# B&R Automation Studio project NAELD004C00R10L518F00 (part 26)

#### Init.st
```iecst
(** 2019-05-20 **)
PROGRAM _INIT

	(* Always Change If Project Change *)

	//Pass Address To Global Address For External Use
	//Action, State & Status
	p_NtParamStat		:= ADR(eStat);
	p_NtParamStatus		:= ADR(eStatus);
	p_NtParamStatTxt	:= ADR(sStatTxt);

	//Alarm
	p_NtParamAlmData	:= ADR(tyAlmData);

	//Output
	p_NtParamFileNotFound				:= ADR(bFileNotFound);

	p_NtParamCurr						:= ADR(tyNtParamCurr);

	p_NtParamDISettings					:= ADR(tyNtParamCurr.tyDISettings);
	p_NtParamDOSettings					:= ADR(tyNtParamCurr.tyDOSettings);
	p_NtParamAWPusherPrep				:= ADR(tyNtParamCurr.bAWPusherPrep);
	p_NtParamAWPrep						:= ADR(tyNtParamCurr.bAWPrep);
	p_NtParamLFPrep						:= ADR(tyNtParamCurr.bLFPrep);
	p_NtParamLeaderMc					:= ADR(tyNtParamCurr.bLeaderMc);
	p_NtParamLFUsrSetPrep				:= ADR(tyNtParamCurr.bLFUsrSetPrep);
	p_NtParamLFWidthLimit				:= ADR(tyNtParamCurr.diLFWidthLimit);
	p_NtParamLFProdWidthChk				:= ADR(tyNtParamCurr.bLFProdWidthChk);
	p_NtParamDSWidthChkPrep				:= ADR(tyNtParamCurr.bDSWidthChkPrep);
	p_NtParamLCSLFPrep					:= ADR(tyNtParamCurr.bLCSLFPrep);
	p_NtParamLCSReqRcpPrep				:= ADR(tyNtParamCurr.bLCSReqRcpPrep);
	p_NtParamLCSManageRcpPrep			:= ADR(tyNtParamCurr.bLCSManageRcpPrep);
	p_NtParamLCSLiveDatPrep				:= ADR(tyNtParamCurr.bLCSLiveDatPrep);
	p_NtParamIPCSMEMA9851ExtdPrep		:= ADR(tyNtParamCurr.bIPCSMEMA9851ExtdPrep);
	p_NtParamVSMEMAPrep					:= ADR(tyNtParamCurr.bVSMEMAPrep);
	p_NtParamHermesPrep					:= ADR(tyNtParamCurr.bHermesPrep);
	p_NtParamHermesRmtPrep				:= ADR(tyNtParamCurr.bHermesRmtPrep);
	p_NtParamSSaverPrep					:= ADR(tyNtParamCurr.bSSaverPrep);
	p_NtParamWidthOffset				:= ADR(tyNtParamCurr.diWidthOffsetInUM);
	p_NtParamPushPulAWidthOffset		:= ADR(tyNtParamCurr.diAWPushPulOffsetInUM);
	p_NtParamJobNo						:= ADR(tyNtParamCurr.sJobNo);
	p_NtParamNtAddr						:= ADR(tyNtParamCurr.usiNtAddr);
	p_NtParamShutterWaitTmr				:= ADR(tyNtParamCurr.tShutterWaitTmr);
	p_NtParamProjAGVInPosSenPrep		:= ADR(tyNtParamCurr.bProjAGVInPosSenPrep);

	p_NtParamProjLaneBPrep				:= ADR(tyNtParamCurr.bProjLaneBPrep);
	p_NtParamProjTopToBtmDefault		:= ADR(tyNtParamCurr.bProjTopToBtmDefault);
	p_NtParamProjLongBrdPrep			:= ADR(tyNtParamCurr.bProjLongBrdPrep);
	p_NtParamProjInletShutPrep			:= ADR(tyNtParamCurr.bProjInletShutPrep);
	p_NtParamProjOutletShutPrep			:= ADR(tyNtParamCurr.bProjOutletShutPrep);
	p_NtParamProjMag1ConvPrep			:= ADR(tyNtParamCurr.bProjMag1ConvPrep);
	p_NtParamProjMag2ConvPrep			:= ADR(tyNtParamCurr.bProjMag2ConvPrep);
	p_NtParamProjMag3ConvPrep			:= ADR(tyNtParamCurr.bProjMag3ConvPrep);
	p_NtParamProjMag4ConvPrep			:= ADR(tyNtParamCurr.bProjMag4ConvPrep);
	p_NtParamProjMagOrientChkSenPrep	:= ADR(tyNtParamCurr.bProjMagOrientChkSenPrep);
	p_NtParamProjAGVPrep				:= ADR(tyNtParamCurr.bProjAGVPrep);
	p_NtParamProjBypsInitConvPrep		:= ADR(tyNtParamCurr.bProjBypsInitConvPrep);
	p_NtParamProjRlsNewProdPrep			:= ADR(tyNtParamCurr.bProjRlsNewProdPrep);
	p_NtParamProjBtnInsertRmvMag		:= ADR(tyNtParamCurr.bProjBtnInsertRmvMag);
	p_NtParamProjMagMinSlt				:= ADR(tyNtParamCurr.diProjMagMinSlt);
	p_NtParamProjMagMaxSlt				:= ADR(tyNtParamCurr.diProjMagMaxSlt);
	p_NtParamProjMag					:= ADR(tyNtParamCurr.eProjMag);
	p_NtParamProjConvDir				:= ADR(tyNtParamCurr.eProjConvDir);
	p_NtParamProjMagConvDir				:= ADR(tyNtParamCurr.eProjMagConvDir);
	p_NtParamProjMagAutoVerifyPrep		:= ADR(tyNtParamCurr.bMagAutoVerifyPrep);
	p_NtParamProjMotorizedPullerPrep	:= ADR(tyNtParamCurr.bProjMotorizedPullerPrep);
	p_NtParamProjMagSafetyBarPrep		:= ADR(tyNtParamCurr.bProjMagSafetyBarPrep);
	p_NtParamProjLifterMagPlatform		:= ADR(tyNtParamCurr.bProjLifterMagPlatform);

	p_NtParamUsrFolderProgNm			:= ADR(tyNtParamCurr.sUsrFolderProgNm);

	p_NtParamLibVersionProgNm			:= ADR(tyNtParamCurr.sLibVersionProgNm);

	p_NtParamTimeProgNm					:= ADR(tyNtParamCurr.sTimeProgNm);

	p_NtParamHWInfoProgNm				:= ADR(tyNtParamCurr.sHWInfoProgNm);
	p_NtParamHWInfoDevice				:= ADR(tyNtParamCurr.sHWInfoDevice);

	p_NtParamTLBuzMode					:= ADR(tyNtParamCurr.eTLBuzMode);

	p_NtParamTLChgRcpBlinkTm		:= ADR(tyNtParamCurr.tTLChgRcpBlinkTm);

	p_NtParamTLErrBlinkTm			:= ADR(tyNtParamCurr.tTLErrBlinkTm);
	p_NtParamBuzErrOnTm				:= ADR(tyNtParamCurr.tBuzErrOnTm);
	p_NtParamBuzErrRestTm			:= ADR(tyNtParamCurr.tBuzErrRestTm);
	p_NtParamBuzErrOnCntr			:= ADR(tyNtParamCurr.usiBuzErrOnCntr);
	p_NtParamBuzErrStopSeqEn		:= ADR(tyNtParamCurr.bBuzErrStopSeqEn);
	p_NtParamBuzErrStopSeqCntr		:= ADR(tyNtParamCurr.usiBuzErrStopSeqCntr);

	p_NtParamTLWarnBlinkTm			:= ADR(tyNtParamCurr.tTLWarnBlinkTm);
	p_NtParamBuzWarnOnTm			:= ADR(tyNtParamCurr.tBuzWarnOnTm);
	p_NtParamBuzWarnRestTm			:= ADR(tyNtParamCurr.tBuzWarnRestTm);
	p_NtParamBuzWarnOnCntr			:= ADR(tyNtParamCurr.usiBuzWarnOnCntr);
	p_NtParamBuzWarnStopSeqEn		:= ADR(tyNtParamCurr.bBuzWarnStopSeqEn);
	p_NtParamBuzWarnStopSeqCntr		:= ADR(tyNtParamCurr.usiBuzWarnStopSeqCntr);

	p_NtParamTLWarn1BlinkTm			:= ADR(tyNtParamCurr.tTLWarn1BlinkTm);
	p_NtParamBuzWarn1OnTm			:= ADR(tyNtParamCurr.tBuzWarn1OnTm);
	p_NtParamBuzWarn1RestTm			:= ADR(tyNtParamCurr.tBuzWarn1RestTm);
	p_NtParamBuzWarn1OnCntr			:= ADR(tyNtParamCurr.usiBuzWarn1OnCntr);
	p_NtParamBuzWarn1StopSeqEn		:= ADR(tyNtParamCurr.bBuzWarn1StopSeqEn);
	p_NtParamBuzWarn1StopSeqCntr	:= ADR(tyNtParamCurr.usiBuzWarn1StopSeqCntr);

	p_NtParamTLWarn2BlinkTm			:= ADR(tyNtParamCurr.tTLWarn2BlinkTm);
	p_NtParamBuzWarn2OnTm			:= ADR(tyNtParamCurr.tBuzWarn2OnTm);
	p_NtParamBuzWarn2RestTm			:= ADR(tyNtParamCurr.tBuzWarn2RestTm);
	p_NtParamBuzWarn2OnCntr			:= ADR(tyNtParamCurr.usiBuzWarn2OnCntr);
	p_NtParamBuzWarn2StopSeqEn		:= ADR(tyNtParamCurr.bBuzWarn2StopSeqEn);
	p_NtParamBuzWarn2StopSeqCntr	:= ADR(tyNtParamCurr.usiBuzWarn2StopSeqCntr);

	p_NtParamTLWarn3BlinkTm			:= ADR(tyNtParamCurr.tTLWarn3BlinkTm);
	p_NtParamBuzWarn3OnTm			:= ADR(tyNtParamCurr.tBuzWarn3OnTm);
	p_NtParamBuzWarn3RestTm			:= ADR(tyNtParamCurr.tBuzWarn3RestTm);
	p_NtParamBuzWarn3OnCntr			:= ADR(tyNtParamCurr.usiBuzWarn3OnCntr);
	p_NtParamBuzWarn3StopSeqEn		:= ADR(tyNtParamCurr.bBuzWarn3StopSeqEn);
	p_NtParamBuzWarn3StopSeqCntr	:= ADR(tyNtParamCurr.usiBuzWarn3StopSeqCntr);

	p_NtParamTLWarn4BlinkTm			:= ADR(tyNtParamCurr.tTLWarn4BlinkTm);
	p_NtParamBuzWarn4OnTm			:= ADR(tyNtParamCurr.tBuzWarn4OnTm);
	p_NtParamBuzWarn4RestTm			:= ADR(tyNtParamCurr.tBuzWarn4RestTm);
	p_NtParamBuzWarn4OnCntr			:= ADR(tyNtParamCurr.usiBuzWarn4OnCntr);
	p_NtParamBuzWarn4StopSeqEn		:= ADR(tyNtParamCurr.bBuzWarn4StopSeqEn);
	p_NtParamBuzWarn4StopSeqCntr	:= ADR(tyNtParamCurr.usiBuzWarn4StopSeqCntr);

	p_NtParamTLWarn5BlinkTm			:= ADR(tyNtParamCurr.tTLWarn5BlinkTm);
	p_NtParamBuzWarn5OnTm			:= ADR(tyNtParamCurr.tBuzWarn5OnTm);
	p_NtParamBuzWarn5RestTm			:= ADR(tyNtParamCurr.tBuzWarn5RestTm);
	p_NtParamBuzWarn5OnCntr			:= ADR(tyNtParamCurr.usiBuzWarn5OnCntr);
	p_NtParamBuzWarn5StopSeqEn		:= ADR(tyNtParamCurr.bBuzWarn5StopSeqEn);
	p_NtParamBuzWarn5StopSeqCntr	:= ADR(tyNtParamCurr.usiBuzWarn5StopSeqCntr);

	p_NtParamBuzAlertOnTm			:= ADR(tyNtParamCurr.tBuzAlertOnTm);
	p_NtParamBuzAlertRestTm			:= ADR(tyNtParamCurr.tBuzAlertRestTm);
	p_NtParamBuzAlertOnCntr			:= ADR(tyNtParamCurr.usiBuzAlertOnCntr);
	p_NtParamBuzAlertStopSeqEn		:= ADR(tyNtParamCurr.bBuzAlertStopSeqEn);
	p_NtParamBuzAlertStopSeqCntr	:= ADR(tyNtParamCurr.usiBuzAlertStopSeqCntr);

	p_NtParamTLBlueBlinkTm			:= ADR(tyNtParamCurr.tTLBlueBlinkTm);
	p_NtParamTLAmberBlinkTm			:= ADR(tyNtParamCurr.tTLAmberBlinkTm);
	p_NtParamTLWhiteBlinkTm			:= ADR(tyNtParamCurr.tTLWhiteBlinkTm);
	p_NtParamTLRedBlinkTm			:= ADR(tyNtParamCurr.tTLRedBlinkTm);
	p_NtParamTLGreenBlinkTm			:= ADR(tyNtParamCurr.tTLGreenBlinkTm);

	p_NtParamAlmProgNm					:= ADR(tyNtParamCurr.sAlmProgNm);
	p_NtParamAlmFileKeepDay				:= ADR(tyNtParamCurr.udiAlmFileKeepDay);

	p_NtParamProdRcpProgNm				:= ADR(tyNtParamCurr.sProdRcpProgNm);
	p_NtParamProdRcpListFileNm			:= ADR(tyNtParamCurr.sProdRcpListFileNm);
	p_NtParamProdRcpSingleFileNm		:= ADR(tyNtParamCurr.sProdRcpSingleFileNm);

	p_NtParamMpProdRcpProgNm			:= ADR(tyNtParamCurr.sMpProdRcpProgNm);
	p_NtParamMpProdRcpFileNm			:= ADR(tyNtParamCurr.sMpProdRcpFileNm);
	p_NtParamMpProdRcpPVNm				:= ADR(tyNtParamCurr.sMpProdRcpPVNm);

	p_NtParamMagRcpProgNm				:= ADR(tyNtParamCurr.sMagRcpProgNm);
	p_NtParamMagRcpListFileNm			:= ADR(tyNtParamCurr.sMagRcpListFileNm);
	p_NtParamMagRcpSingleFileNm			:= ADR(tyNtParamCurr.sMagRcpSingleFileNm);

	p_NtParamMagRcpProgNm1				:= ADR(tyNtParamCurr.sMagRcpProgNm1);
	p_NtParamMagRcpListFileNm1			:= ADR(tyNtParamCurr.sMagRcpListFileNm1);
	p_NtParamMagRcpSingleFileNm1		:= ADR(tyNtParamCurr.sMagRcpSingleFileNm1);

	p_NtParamMcParamProgNm				:= ADR(tyNtParamCurr.sMcParamProgNm);
	p_NtParamMcParamFileNm				:= ADR(tyNtParamCurr.sMcParamFileNm);

	p_NtParamUsrMgmtProgNm				:= ADR(tyNtParamCurr.sUsrMgmtProgNm);

	p_NtParamBffr1ProgNm				:= ADR(tyNtParamCurr.sBffr1ProgNm);
	p_NtParamBffr1FileNm				:= ADR(tyNtParamCurr.sBffr1FileNm);
	p_NtParamBffr1FIFO					:= ADR(tyNtParamCurr.bBffr1FIFO);

	p_NtParamBffr2ProgNm				:= ADR(tyNtParamCurr.sBffr2ProgNm);
	p_NtParamBffr2FileNm				:= ADR(tyNtParamCurr.sBffr2FileNm);
	p_NtParamBffr2FIFO					:= ADR(tyNtParamCurr.bBffr2FIFO);

	p_NtParamBffr3ProgNm				:= ADR(tyNtParamCurr.sBffr3ProgNm);
	p_NtParamBffr3FileNm				:= ADR(tyNtParamCurr.sBffr3FileNm);
	p_NtParamBffr3FIFO					:= ADR(tyNtParamCurr.bBffr3FIFO);

	p_NtParamBffr4ProgNm				:= ADR(tyNtParamCurr.sBffr4ProgNm);
	p_NtParamBffr4FileNm				:= ADR(tyNtParamCurr.sBffr4FileNm);
	p_NtParamBffr4FIFO					:= ADR(tyNtParamCurr.bBffr4FIFO);

	p_NtParamUSSMEMA1ProgNm				:= ADR(tyNtParamCurr.sUSSMEMA1ProgNm);
	p_NtParamUSSMEMA1RstDlyTm			:= ADR(tyNtParamCurr.tUSSMEMA1RstDlyTm);
	p_NtParamUSSMEMA1SigInChkTm			:= ADR(tyNtParamCurr.tUSSMEMA1SigInChkTm);

	p_NtParamUSSMEMA2ProgNm				:= ADR(tyNtParamCurr.sUSSMEMA2ProgNm);
	p_NtParamUSSMEMA2RstDlyTm			:= ADR(tyNtParamCurr.tUSSMEMA2RstDlyTm);
	p_NtParamUSSMEMA2SigInChkTm			:= ADR(tyNtParamCurr.tUSSMEMA2SigInChkTm);

	p_NtParamUSSMEMA3ProgNm				:= ADR(tyNtParamCurr.sUSSMEMA3ProgNm);
	p_NtParamUSSMEMA3RstDlyTm			:= ADR(tyNtParamCurr.tUSSMEMA3RstDlyTm);
	p_NtParamUSSMEMA3SigInChkTm			:= ADR(tyNtParamCurr.tUSSMEMA3SigInChkTm);

	p_NtParamUSSMEMA4ProgNm				:= ADR(tyNtParamCurr.sUSSMEMA4ProgNm);
	p_NtParamUSSMEMA4RstDlyTm			:= ADR(tyNtParamCurr.tUSSMEMA4RstDlyTm);
	p_NtParamUSSMEMA4SigInChkTm			:= ADR(tyNtParamCurr.tUSSMEMA4SigInChkTm);

	p_NtParamDSSMEMA1ProgNm				:= ADR(tyNtParamCurr.sDSSMEMA1ProgNm);
	p_NtParamDSSMEMA1RstDlyTm			:= ADR(tyNtParamCurr.tDSSMEMA1RstDlyTm);
	p_NtParamDSSMEMA1SigInChkTm			:= ADR(tyNtParamCurr.tDSSMEMA1SigInChkTm);

	p_NtParamDSSMEMA2ProgNm				:= ADR(tyNtParamCurr.sDSSMEMA2ProgNm);
	p_NtParamDSSMEMA2RstDlyTm			:= ADR(tyNtParamCurr.tDSSMEMA2RstDlyTm);
	p_NtParamDSSMEMA2SigInChkTm			:= ADR(tyNtParamCurr.tDSSMEMA2SigInChkTm);

	p_NtParamDSSMEMA3ProgNm				:= ADR(tyNtParamCurr.sDSSMEMA3ProgNm);
	p_NtParamDSSMEMA3RstDlyTm			:= ADR(tyNtParamCurr.tDSSMEMA3RstDlyTm);
	p_NtParamDSSMEMA3SigInChkTm			:= ADR(tyNtParamCurr.tDSSMEMA3SigInChkTm);

	p_NtParamDSSMEMA4ProgNm				:= ADR(tyNtParamCurr.sDSSMEMA4ProgNm);
	p_NtParamDSSMEMA4RstDlyTm			:= ADR(tyNtParamCurr.tDSSMEMA4RstDlyTm);
	p_NtParamDSSMEMA4SigInChkTm			:= ADR(tyNtParamCurr.tDSSMEMA4SigInChkTm);

	p_NtParamDSSMEMAAProgNm				:= ADR(tyNtParamCurr.sDSSMEMAAProgNm);
	p_NtParamDSSMEMAARstDlyTm			:= ADR(tyNtParamCurr.tDSSMEMAARstDlyTm);
	p_NtParamDSSMEMAASigInChkTm			:= ADR(tyNtParamCurr.tDSSMEMAASigInChkTm);

	p_NtParamDSSMEMABProgNm				:= ADR(tyNtParamCurr.sDSSMEMABProgNm);
	p_NtParamDSSMEMABRstDlyTm			:= ADR(tyNtParamCurr.tDSSMEMABRstDlyTm);
	p_NtParamDSSMEMABSigInChkTm			:= ADR(tyNtParamCurr.tDSSMEMABSigInChkTm);

	p_NtParamInShutterProgNm			:= ADR(tyNtParamCurr.sInShutterProgNm);
	p_NtParamInShutterTwoCtrlIn			:= ADR(tyNtParamCurr.bInShutterTwoCtrlIn);
	p_NtParamInShutterExtTO				:= ADR(tyNtParamCurr.tInShutterExtTO);
	p_NtParamInShutterRetTO				:= ADR(tyNtParamCurr.tInShutterRetTO);

	p_NtParamOutShutterProgNm			:= ADR(tyNtParamCurr.sOutShutterProgNm);
	p_NtParamOutShutterTwoCtrlIn		:= ADR(tyNtParamCurr.bOutShutterTwoCtrlIn);
	p_NtParamOutShutterExtTO			:= ADR(tyNtParamCurr.tOutShutterExtTO);
	p_NtParamOutShutterRetTO			:= ADR(tyNtParamCurr.tOutShutterRetTO);

	p_NtParamPullConvProgNm				:= ADR(tyNtParamCurr.sPullConvProgNm);
	p_NtParamPullConvOnDirMod			:= ADR(tyNtParamCurr.bPullConvOnDirMod);
	p_NtParamPullConvMtrOffDlyTm		:= ADR(tyNtParamCurr.tPullConvMtrOffDlyTm);
	p_NtParamPullConvPullExtTO			:= ADR(tyNtParamCurr.tPullConvPullExtTO);
	p_NtParamPullConvPullRetTO			:= ADR(tyNtParamCurr.tPullConvPullRetTO);
	p_NtParamPullConvRotHomeTO			:= ADR(tyNtParamCurr.tPullConvRotHomeTO);
	p_NtParamPullConvRotRemoteTO		:= ADR(tyNtParamCurr.tPullConvRotRemoteTO);

	p_NtParamMagConv1ProgNm				:= ADR(tyNtParamCurr.sMagConv1ProgNm);
	p_NtParamMagConv1OnDirMod			:= ADR(tyNtParamCurr.bMagConv1OnDirMod);
	p_NtParamMagConv1MtrOffDlyTm		:= ADR(tyNtParamCurr.tMagConv1MtrOffDlyTm);
	p_NtParamMagConv1ClprClampTO		:= ADR(tyNtParamCurr.tMagConv1ClprClampTO);
	p_NtParamMagConv1ClprUnclampTO		:= ADR(tyNtParamCurr.tMagConv1ClprUnclampTO);

	p_NtParamMagConv2ProgNm				:= ADR(tyNtParamCurr.sMagConv2ProgNm);
	p_NtParamMagConv2OnDirMod			:= ADR(tyNtParamCurr.bMagConv2OnDirMod);
	p_NtParamMagConv2MtrOffDlyTm		:= ADR(tyNtParamCurr.tMagConv2MtrOffDlyTm);
	p_NtParamMagConv2ClprClampTO		:= ADR(tyNtParamCurr.tMagConv2ClprClampTO);
	p_NtParamMagConv2ClprUnclampTO		:= ADR(tyNtParamCurr.tMagConv2ClprUnclampTO);

	p_NtParamMagConv3ProgNm				:= ADR(tyNtParamCurr.sMagConv3ProgNm);
	p_NtParamMagConv3OnDirMod			:= ADR(tyNtParamCurr.bMagConv3OnDirMod);
	p_NtParamMagConv3MtrOffDlyTm		:= ADR(tyNtParamCurr.tMagConv3MtrOffDlyTm);
	p_NtParamMagConv3ClprClampTO		:= ADR(tyNtParamCurr.tMagConv3ClprClampTO);
	p_NtParamMagConv3ClprUnclampTO		:= ADR(tyNtParamCurr.tMagConv3ClprUnclampTO);

	p_NtParamMagConv4ProgNm				:= ADR(tyNtParamCurr.sMagConv4ProgNm);
	p_NtParamMagConv4OnDirMod			:= ADR(tyNtParamCurr.bMagConv4OnDirMod);
	p_NtParamMagConv4MtrOffDlyTm		:= ADR(tyNtParamCurr.tMagConv4MtrOffDlyTm);
	p_NtParamMagConv4ClprClampTO		:= ADR(tyNtParamCurr.tMagConv4ClprClampTO);
	p_NtParamMagConv4ClprUnclampTO		:= ADR(tyNtParamCurr.tMagConv4ClprUnclampTO);

	p_NtParamMtrPshrProgNm				:= ADR(tyNtParamCurr.sMtrPshrProgNm);
	p_NtParamMtrPshrDir					:= ADR(tyNtParamCurr.bMtrPshrDir);
	p_NtParamMtrPshrAlmRstTm			:= ADR(tyNtParamCurr.tMtrPshrAlmRstTm);
	p_NtParamMtrPshrAlmTrigTm			:= ADR(tyNtParamCurr.tMtrPshrAlmTrigTm);
	p_NtParamMtrPshrExtTO				:= ADR(tyNtParamCurr.tMtrPshrExtTO);
	p_NtParamMtrPshrRetTO				:= ADR(tyNtParamCurr.tMtrPshrRetTO);
	p_NtParamMtrPshrExtSlowSpd			:= ADR(tyNtParamCurr.diMtrPshrExtSlowSpd);
	p_NtParamMtrPshrRetSlowSpd			:= ADR(tyNtParamCurr.diMtrPshrRetSlowSpd);
	p_NtParamMtrPshrExtNomSpd			:= ADR(tyNtParamCurr.diMtrPshrExtNomSpd);
	p_NtParamMtrPshrExtTorq				:= ADR(tyNtParamCurr.diMtrPshrExtTorq);
	p_NtParamMtrPshrRetTorq				:= ADR(tyNtParamCurr.diMtrPshrRetTorq);
	p_NtParamMtrPshrStartTorq			:= ADR(tyNtParamCurr.diMtrPshrStartTorq);

	p_NtParamAWPushPulProgNm			:= ADR(tyNtParamCurr.sAWPushPullProgNm);
	p_NtParamAWPushPulDevice			:= ADR(tyNtParamCurr.sAWPushPullDevice);
	p_NtParamAWPushPulNode				:= ADR(tyNtParamCurr.usiAWPushPullNode);
	p_NtParamAWPushPulDir				:= ADR(tyNtParamCurr.bAWPushPullDir);
	p_NtParamAWPushPulDirBl				:= ADR(tyNtParamCurr.bAWPushPullDirBl);
	p_NtParamAWPushPulPitchInUM			:= ADR(tyNtParamCurr.diAWPushPullPitchInUM);
	p_NtParamAWPushPulMovBlDistInUM		:= ADR(tyNtParamCurr.diAWPushPullMovBlDistInUM);
	p_NtParamAWPushPulParamInHm			:= ADR(tyNtParamCurr.tyAWPushPullParamInHm);
	p_NtParamAWPushPulParamInConvert	:= ADR(tyNtParamCurr.tyAWPushPullParamInConvert);
	p_NtParamAWPushPulParam				:= ADR(tyNtParamCurr.tyAWPushPullParam);
	p_NtParamAWPushPulAcc				:= ADR(tyNtParamCurr.tyAWPushPullParam.diAccInMS);
	p_NtParamAWPushPulDec				:= ADR(tyNtParamCurr.tyAWPushPullParam.diDecInMS);
	p_NtParamAWPushPulAutoSpd			:= ADR(tyNtParamCurr.tyAWPushPullParam.diAutoSpdInUMPS);
	p_NtParamAWPushPulTuning			:= ADR(tyNtParamCurr.tyAWPushPullTuning);
	p_NtParamAWPushPulMotorType			:= ADR(tyNtParamCurr.eAWPushPullServoMotorType);

	p_NtParamAWProgNm					:= ADR(tyNtParamCurr.sAWProgNm);
	p_NtParamAWDevice					:= ADR(tyNtParamCurr.sAWDevice);
	p_NtParamAWNode						:= ADR(tyNtParamCurr.usiAWNode);
	p_NtParamAWDir						:= ADR(tyNtParamCurr.bAWDir);
	p_NtParamAWDirBl					:= ADR(tyNtParamCurr.bAWDirBl);
	p_NtParamAWPitchInUM				:= ADR(tyNtParamCurr.diAWPitchInUM);
	p_NtParamAWMovBlDistInUM			:= ADR(tyNtParamCurr.diAWMovBlDistInUM);
	p_NtParamAWParamInHm				:= ADR(tyNtParamCurr.tyAWParamInHm);
	p_NtParamAWParamInConvert			:= ADR(tyNtParamCurr.tyAWParamInConvert);
	p_NtParamAWParam					:= ADR(tyNtParamCurr.tyAWParam);
	p_NtParamAWAcc						:= ADR(tyNtParamCurr.tyAWParam.diAccInMS);
	p_NtParamAWDec						:= ADR(tyNtParamCurr.tyAWParam.diDecInMS);
	p_NtParamAWAutoSpd					:= ADR(tyNtParamCurr.tyAWParam.diAutoSpdInUMPS);
	p_NtParamAWTuning					:= ADR(tyNtParamCurr.tyAWTuning);
	p_NtParamAWMotorType				:= ADR(tyNtParamCurr.eAWServoMotorType);

	p_NtParamTravProgNm					:= ADR(tyNtParamCurr.sTravProgNm);
	p_NtParamTravDevice					:= ADR(tyNtParamCurr.sTravDevice);
	p_NtParamTravNode					:= ADR(tyNtParamCurr.usiTravNode);
	p_NtParamTravDir					:= ADR(tyNtParamCurr.bTravDir);
	p_NtParamTravParamInHm				:= ADR(tyNtParamCurr.tyTravParamInHm);
	p_NtParamTravParamInConvert			:= ADR(tyNtParamCurr.tyTravParamInConvert);
	p_NtParamTravParam					:= ADR(tyNtParamCurr.tyTravParam);
	p_NtParamTravAcc					:= ADR(tyNtParamCurr.tyTravParam.diAccInMS);
	p_NtParamTravDec					:= ADR(tyNtParamCurr.tyTravParam.diDecInMS);
	p_NtParamTravAutoSpd				:= ADR(tyNtParamCurr.tyTravParam.diAutoSpdInUMPS);
	p_NtParamTravTuning					:= ADR(tyNtParamCurr.tyTravTuning);
	p_NtParamTravLongBrdAutoSpd			:= ADR(tyNtParamCurr.diTravAutoSpdLongBrdInUMPS);
	p_NtParamTravMotorType				:= ADR(tyNtParamCurr.eTravServoMotorType);

	p_NtParamLifterProgNm				:= ADR(tyNtParamCurr.sLifterProgNm);
	p_NtParamLifterDevice				:= ADR(tyNtParamCurr.sLifterDevice);
	p_NtParamLifterNode					:= ADR(tyNtParamCurr.usiLifterNode);
	p_NtParamLifterDir					:= ADR(tyNtParamCurr.bLifterDir);
	p_NtParamLifterParamInHm			:= ADR(tyNtParamCurr.tyLifterParamInHm);
	p_NtParamLifterParamInConvert		:= ADR(tyNtParamCurr.tyLifterParamInConvert);
	p_NtParamLifterParam				:= ADR(tyNtParamCurr.tyLifterParam);
	p_NtParamLifterAcc					:= ADR(tyNtParamCurr.tyLifterParam.diAccInMS);
	p_NtParamLifterDec					:= ADR(tyNtParamCurr.tyLifterParam.diDecInMS);
	p_NtParamLifterAutoSpd				:= ADR(tyNtParamCurr.tyLifterParam.diAutoSpdInUMPS);
	p_NtParamLifterTuning				:= ADR(tyNtParamCurr.tyLifterTuning);
	p_NtParamLifterMotorType			:= ADR(tyNtParamCurr.eLifterServoMotorType);

	p_NtParamDIProgNm					:= ADR(tyNtParamCurr.sDIProgNm);

	p_NtParamAIVSvrProgNm				:= ADR(tyNtParamCurr.sAGVSvrProgNm);

	p_NtParamAGVMag1ProgNm				:= ADR(tyNtParamCurr.sAGVMag1ProgNm);
	p_NtParamAGVMag2ProgNm				:= ADR(tyNtParamCurr.sAGVMag2ProgNm);
	p_NtParamAGVMag3ProgNm				:= ADR(tyNtParamCurr.sAGVMag3ProgNm);
	p_NtParamAGVMag4ProgNm				:= ADR(tyNtParamCurr.sAGVMag4ProgNm);

	p_NtParamHermesProgNm				:= ADR(tyNtParamCurr.sHermesProgNm);
	p_NtParamHermesRetainFileNm			:= ADR(tyNtParamCurr.sHermesRetainFileNm);
	p_NtParamHermesConfigFileNm			:= ADR(tyNtParamCurr.sHermesConfigFileNm);

	p_NtParamDSHermesAProgNm			:= ADR(tyNtParamCurr.sDSHermesAProgNm);
	p_NtParamDSHermesAFileKeepDay		:= ADR(tyNtParamCurr.udiDSHermesAFileKeepDay);
	p_NtParamDSHermesAAliveTmInSec		:= ADR(tyNtParamCurr.udiDSHermesAAliveTmInSec);
	p_NtParamDSHermesAConnTO			:= ADR(tyNtParamCurr.tDSHermesAConnTO);

	p_NtParamDSHermesBProgNm			:= ADR(tyNtParamCurr.sDSHermesBProgNm);
	p_NtParamDSHermesBFileKeepDay		:= ADR(tyNtParamCurr.udiDSHermesBFileKeepDay);
	p_NtParamDSHermesBAliveTmInSec		:= ADR(tyNtParamCurr.udiDSHermesBAliveTmInSec);
	p_NtParamDSHermesBConnTO			:= ADR(tyNtParamCurr.tDSHermesBConnTO);

	p_NtParamRmtHermesProgNm			:= ADR(tyNtParamCurr.sRmtHermesProgNm);
	p_NtParamRmtHermesConfigFileNm		:= ADR(tyNtParamCurr.sRmtHermesConfigFileNm);
	p_NtParamRmtHermesFileKeepDay		:= ADR(tyNtParamCurr.udiRmtHermesFileKeepDay);
	p_NtParamRmtHermesAliveTmInSec		:= ADR(tyNtParamCurr.udiRmtHermesAliveTmInSec);
	p_NtParamRmtHermesSndBffrSize		:= ADR(tyNtParamCurr.udiRmtHermesSndBffrSize);
	p_NtParamRmtHermesRcvBffrSize		:= ADR(tyNtParamCurr.udiRmtHermesRcvBffrSize);

	p_NtParamLFLeaderProgNm				:= ADR(tyNtParamCurr.sLFLeaderProgNm);
	p_NtParamLFLeaderOnlineChkDlyTm		:= ADR(tyNtParamCurr.tLFLeaderOnlineChkDlyTm);
	p_NtParamLFLeaderSetTmOffDlyTm		:= ADR(tyNtParamCurr.tLFLeaderSetTmOffDlyTm);

	p_NtParamLFFollowerProgNm			:= ADR(tyNtParamCurr.sLFFollowerProgNm);

	p_NtParamFollower1ProgNm			:= ADR(tyNtParamCurr.sFollower1ProgNm);
	p_NtParamFollower2ProgNm			:= ADR(tyNtParamCurr.sFollower2ProgNm);

	p_NtParamLCSProgNm					:= ADR(tyNtParamCurr.sLCSProgNm);

	p_NtParamLCSMngRcpProgNm			:= ADR(tyNtParamCurr.sLCSMngRcpProgNm);

	p_NtParamLCSLFProgNm				:= ADR(tyNtParamCurr.sLCSLFProgNm);

	p_NtParamOpsTravLifLDProgNm			:= ADR(tyNtParamCurr.sOpsTravLifLDProgNm);

	p_NtParamOpsMagLD1ProgNm			:= ADR(tyNtParamCurr.sOpsMagLD1ProgNm);

	p_NtParamOpsMagLD2ProgNm			:= ADR(tyNtParamCurr.sOpsMagLD2ProgNm);

	p_NtParamOpsMagLD3ProgNm			:= ADR(tyNtParamCurr.sOpsMagLD3ProgNm);

	p_NtParamOpsMagLD4ProgNm			:= ADR(tyNtParamCurr.sOpsMagLD4ProgNm);

	p_NtParamOpsMagConvLD1ProgNm		:= ADR(tyNtParamCurr.sOpsMagConvLD1ProgNm);

	p_NtParamOpsMagConvLD2ProgNm		:= ADR(tyNtParamCurr.sOpsMagConvLD2ProgNm);

	p_NtParamOpsMagConvLD3ProgNm		:= ADR(tyNtParamCurr.sOpsMagConvLD3ProgNm);

	p_NtParamOpsMagConvLD4ProgNm		:= ADR(tyNtParamCurr.sOpsMagConvLD4ProgNm);

	p_NtParamOpsLifMagLDProgNm			:= ADR(tyNtParamCurr.sOpsLifMagLDProgNm);

	p_NtParamProdRcpMinWidth			:= ADR(tyNtParamCurr.tyProdRcpWidth.diMin);
	p_NtParamProdRcpMaxWidth			:= ADR(tyNtParamCurr.tyProdRcpWidth.diMax);
	p_NtParamProdRcpMinMinSlt			:= ADR(tyNtParamCurr.tyProdRcpMinSlt.diMin);
	p_NtParamProdRcpMaxMinSlt			:= ADR(tyNtParamCurr.tyProdRcpMinSlt.diMax);
	p_NtParamProdRcpMinMaxSlt			:= ADR(tyNtParamCurr.tyProdRcpMaxSlt.diMin);
	p_NtParamProdRcpMaxMaxSlt			:= ADR(tyNtParamCurr.tyProdRcpMaxSlt.diMax);
	p_NtParamProdRcpMinPitch			:= ADR(tyNtParamCurr.tyProdRcpPitch.diMin);
	p_NtParamProdRcpMaxPitch			:= ADR(tyNtParamCurr.tyProdRcpPitch.diMax);
	p_NtParamProdRcpMinMcModA			:= ADR(tyNtParamCurr.tyProdRcpMcModA.diMin);
	p_NtParamProdRcpMaxMcModA			:= ADR(tyNtParamCurr.tyProdRcpMcModA.diMax);
	p_NtParamProdRcpMinMcModAB			:= ADR(tyNtParamCurr.tyProdRcpMcModAB.diMin);
	p_NtParamProdRcpMaxMcModAB			:= ADR(tyNtParamCurr.tyProdRcpMcModAB.diMax);

	p_NtParamPullerProgNm				:= ADR(tyNtParamCurr.sPullerProgNm);
	p_NtParamPullerTwoCtrlIn			:= ADR(tyNtParamCurr.bPullerTwoCtrlIn);
	p_NtParamPullerExtTO				:= ADR(tyNtParamCurr.tPullerExtTO);
	p_NtParamPullerRetTO				:= ADR(tyNtParamCurr.tPullerRetTO);
	p_NtParamProjPullerRotCylPrep		:= ADR(tyNtParamCurr.bProjPullerRotCylPrep);
	p_NtParamProjPullerExtMaxSlt		:= ADR(tyNtParamCurr.diProjPullerExtMaxSlt);
	p_NtParamProjPullerExtMinSlt		:= ADR(tyNtParamCurr.diProjPullerExtMinSlt);

	p_NtParamSelClamp1ProgNm			:= ADR(tyNtParamCurr.sSelClamp1ProgNm);
	p_NtParamSelClamp1TwoCtrlIn			:= ADR(tyNtParamCurr.bSelClamp1TwoCtrlIn);
	p_NtParamSelClamp1ExtDlyTm			:= ADR(tyNtParamCurr.tSelClamp1ExtDlyTm);
	p_NtParamSelClamp1RetDlyTm			:= ADR(tyNtParamCurr.tSelClamp1RetDlyTm);

	p_NtParamSelClamp2ProgNm			:= ADR(tyNtParamCurr.sSelClamp2ProgNm);
	p_NtParamSelClamp2TwoCtrlIn			:= ADR(tyNtParamCurr.bSelClamp2TwoCtrlIn);
	p_NtParamSelClamp2ExtDlyTm			:= ADR(tyNtParamCurr.tSelClamp2ExtDlyTm);
	p_NtParamSelClamp2RetDlyTm			:= ADR(tyNtParamCurr.tSelClamp2RetDlyTm);

	p_NtParamSelClamp3ProgNm			:= ADR(tyNtParamCurr.sSelClamp3ProgNm);
	p_NtParamSelClamp3TwoCtrlIn			:= ADR(tyNtParamCurr.bSelClamp3TwoCtrlIn);
	p_NtParamSelClamp3ExtDlyTm			:= ADR(tyNtParamCurr.tSelClamp3ExtDlyTm);
	p_NtParamSelClamp3RetDlyTm			:= ADR(tyNtParamCurr.tSelClamp3RetDlyTm);

	p_NtParamSelClamp4ProgNm			:= ADR(tyNtParamCurr.sSelClamp4ProgNm);
	p_NtParamSelClamp4TwoCtrlIn			:= ADR(tyNtParamCurr.bSelClamp4TwoCtrlIn);
	p_NtParamSelClamp4ExtDlyTm			:= ADR(tyNtParamCurr.tSelClamp4ExtDlyTm);
	p_NtParamSelClamp4RetDlyTm			:= ADR(tyNtParamCurr.tSelClamp4RetDlyTm);

	p_NtParamProjDBAOnRgtSen			:= ADR (tyNtParamCurr.bProjDBAOnRgtSen);

	p_NtParamLFWidth2Prep				:= ADR(tyNtParamCurr.bLFProdWidth2Prep);
	p_NtParamLFFllowerOnlineChkDlyTm	:= ADR(tyNtParamCurr.tLFFollowerOnlineChkDlyTm);

	p_NtParamUSSOT1ProgNm				:= ADR(tyNtParamCurr.sUSSOT1ProgNm);
	p_NtParamUSSOT1RstDlyTm				:= ADR(tyNtParamCurr.tUSSOT1RstDlyTm);
	p_NtParamUSSOT1SigInChkTm			:= ADR(tyNtParamCurr.tUSSOT1SigInChkTm);

	p_NtParamUSSOT2ProgNm				:= ADR(tyNtParamCurr.sUSSOT2ProgNm);
	p_NtParamUSSOT2RstDlyTm				:= ADR(tyNtParamCurr.tUSSOT2RstDlyTm);
	p_NtParamUSSOT2SigInChkTm			:= ADR(tyNtParamCurr.tUSSOT2SigInChkTm);

	p_NtParamUSSOT3ProgNm				:= ADR(tyNtParamCurr.sUSSOT3ProgNm);
	p_NtParamUSSOT3RstDlyTm				:= ADR(tyNtParamCurr.tUSSOT3RstDlyTm);
	p_NtParamUSSOT3SigInChkTm			:= ADR(tyNtParamCurr.tUSSOT3SigInChkTm);

	p_NtParamUSSOT4ProgNm				:= ADR(tyNtParamCurr.sUSSOT4ProgNm);
	p_NtParamUSSOT4RstDlyTm				:= ADR(tyNtParamCurr.tUSSOT4RstDlyTm);
	p_NtParamUSSOT4SigInChkTm			:= ADR(tyNtParamCurr.tUSSOT4SigInChkTm);

	p_NtParamDSSOT1ProgNm				:= ADR(tyNtParamCurr.sDSSOT1ProgNm);
	p_NtParamDSSOT1RstDlyTm				:= ADR(tyNtParamCurr.tDSSOT1RstDlyTm);
	p_NtParamDSSOT1SigInChkTm			:= ADR(tyNtParamCurr.tDSSOT1SigInChkTm);

	p_NtParamDSSOT2ProgNm				:= ADR(tyNtParamCurr.sDSSOT2ProgNm);
	p_NtParamDSSOT2RstDlyTm				:= ADR(tyNtParamCurr.tDSSOT2RstDlyTm);
	p_NtParamDSSOT2SigInChkTm			:= ADR(tyNtParamCurr.tDSSOT2SigInChkTm);

	p_NtParamDSSOT3ProgNm				:= ADR(tyNtParamCurr.sDSSOT3ProgNm);
	p_NtParamDSSOT3RstDlyTm				:= ADR(tyNtParamCurr.tDSSOT3RstDlyTm);
	p_NtParamDSSOT3SigInChkTm			:= ADR(tyNtParamCurr.tDSSOT3SigInChkTm);

	p_NtParamDSSOT4ProgNm				:= ADR(tyNtParamCurr.sDSSOT4ProgNm);
	p_NtParamDSSOT4RstDlyTm				:= ADR(tyNtParamCurr.tDSSOT4RstDlyTm);
	p_NtParamDSSOT4SigInChkTm			:= ADR(tyNtParamCurr.tDSSOT4SigInChkTm);

	p_NtParamProjSOTSenPrep				:= ADR(tyNtParamCurr.bProjSOTSensorPrep);

	p_NtParamMcProgNm					:= ADR(tyNtParamCurr.sMachineProgNm);
	p_NtParamMc1ProgNm					:= ADR(tyNtParamCurr.sMachine1ProgNm);

	p_NtParamProjUSBPrep				:= ADR(tyNtParamCurr.bUSBScannerPrep);
	p_NtParamUSBProgNm					:= ADR(tyNtParamCurr.sUSBRdrProgNm);

	p_NtParamSOTReadyOnFirst			:= ADR(tyNtParamCurr.bSOTReadyOnFirst);

	p_NtParamShowMESName				:= ADR(tyNtParamCurr.bShowMESName);
	p_NtParamShowFMorMESActive			:= ADR(tyNtParamCurr.bShowFMorMESActive);

	p_NtParamRS232Prep					:= ADR(tyNtParamCurr.bRS232ScannerPrep);
	p_NtParamRS232ProgNm				:= ADR(tyNtParamCurr.sRS232ProgNm);

	p_NtParamProdRcpMinMtrPshrExtSpd	:= ADR(tyNtParamCurr.tyProdRcpMtrPshrExtSpd.diMin);
	p_NtParamProdRcpMaxMtrPshrExtSpd	:= ADR(tyNtParamCurr.tyProdRcpMtrPshrExtSpd.diMax);
	p_NtParamProdRcpMinMtrPshrExtToq	:= ADR(tyNtParamCurr.tyProdRcpMtrPshrExtTorq.diMin);
	p_NtParamProdRcpMaxMtrPshrExtToq	:= ADR(tyNtParamCurr.tyProdRcpMtrPshrExtTorq.diMax);

	p_NtParamMag1SafetyBarProgNm		:= ADR(tyNtParamCurr.sMag1SafetyBarProgNm);
	p_NtParamMag1SafetyBarTwoCtrlIn		:= ADR(tyNtParamCurr.bMag1SafetyBarTwoCtrlIn);
	p_NtParamMag1SafetyBarExtTO			:= ADR(tyNtParamCurr.tMag1SafetyBarExtTO);
	p_NtParamMag1SafetyBarRetTO			:= ADR(tyNtParamCurr.tMag1SafetyBarRetTO);

	p_NtParamMag2SafetyBarProgNm		:= ADR(tyNtParamCurr.sMag2SafetyBarProgNm);
	p_NtParamMag2SafetyBarTwoCtrlIn		:= ADR(tyNtParamCurr.bMag2SafetyBarTwoCtrlIn);
	p_NtParamMag2SafetyBarExtTO			:= ADR(tyNtParamCurr.tMag2SafetyBarExtTO);
	p_NtParamMag2SafetyBarRetTO			:= ADR(tyNtParamCurr.tMag2SafetyBarRetTO);

	p_NtParamMag3SafetyBarProgNm		:= ADR(tyNtParamCurr.sMag3SafetyBarProgNm);
	p_NtParamMag3SafetyBarTwoCtrlIn		:= ADR(tyNtParamCurr.bMag3SafetyBarTwoCtrlIn);
	p_NtParamMag3SafetyBarExtTO			:= ADR(tyNtParamCurr.tMag3SafetyBarExtTO);
	p_NtParamMag3SafetyBarRetTO			:= ADR(tyNtParamCurr.tMag3SafetyBarRetTO);

	p_NtParamMag4SafetyBarProgNm		:= ADR(tyNtParamCurr.sMag4SafetyBarProgNm);
	p_NtParamMag4SafetyBarTwoCtrlIn		:= ADR(tyNtParamCurr.bMag4SafetyBarTwoCtrlIn);
	p_NtParamMag4SafetyBarExtTO			:= ADR(tyNtParamCurr.tMag4SafetyBarExtTO);
	p_NtParamMag4SafetyBarRetTO			:= ADR(tyNtParamCurr.tMag4SafetyBarRetTO);

	p_NtParamPullerHeightInMM			:= ADR(tyNtParamCurr.diPullerHeightInMM);

	p_NtParamProjDsFixToFixRail		:= ADR(tyNtParamCurr.bProjDSFixToFixRail);
	p_NtParamProjWorkOrderOPCUA		:= ADR(tyNtParamCurr.bProjWorkOrderOPCUA);

	p_NtParamProjServoPullPusherPrep	:= ADR(tyNtParamCurr.bProjServoPullerPusherPrep);
	p_NtParamPPProgNm					:= ADR(tyNtParamCurr.sPPProgNm);
	p_NtParamPPDevice					:= ADR(tyNtParamCurr.sPPDevice);
	p_NtParamPPNode						:= ADR(tyNtParamCurr.usiPPNode);
	p_NtParamPPDir						:= ADR(tyNtParamCurr.bPPDir);
	p_NtParamPPDirBl					:= ADR(tyNtParamCurr.bPPDirBl);
	p_NtParamPPPitchInUM				:= ADR(tyNtParamCurr.diPPPitchInUM);
	p_NtParamPPMovBlDistInUM			:= ADR(tyNtParamCurr.diPPMovBlDistInUM);
	p_NtParamPPParamInHm				:= ADR(tyNtParamCurr.tyPPParamInHm);
	p_NtParamPPParamInConvert			:= ADR(tyNtParamCurr.tyPPParamInConvert);
	p_NtParamPPParam					:= ADR(tyNtParamCurr.tyPPParam);
	p_NtParamPPAcc						:= ADR(tyNtParamCurr.tyPPParam.diAccInMS);
	p_NtParamPPDec						:= ADR(tyNtParamCurr.tyPPParam.diDecInMS);
	p_NtParamPPAutoSpd					:= ADR(tyNtParamCurr.tyPPParam.diAutoSpdInUMPS);
	p_NtParamPPTuning					:= ADR(tyNtParamCurr.tyPPTuning);
	p_NtParamPPMotorType				:= ADR(tyNtParamCurr.ePPServoMotorType);

	p_NtParamProjCurtainSenPrep			:= ADR(tyNtParamCurr.bProjCurtainSenPrep);
	p_NtParamProjMagHeightChkPrep		:= ADR(tyNtParamCurr.bProjMagHeightChkPrep);
	p_NtParamTravGotoMagWidthChkPt1		:= ADR(tyNtParamCurr.diTravGoToMagWidthChkPt1);
	p_NtParamTravGotoMagWidthChkPt2		:= ADR(tyNtParamCurr.diTravGoToMagWidthChkPt2);
	p_NtParamTravGotoMagWidthChkPt3		:= ADR(tyNtParamCurr.diTravGoToMagWidthChkPt3);

	p_NtParamPPTorqParam				:= ADR(tyNtParamCurr.tyPPTorqParam);
	p_NtParamProjLifTravMnlLoad			:= ADR(tyNtParamCurr.bProjLifTravMnlLoad);
	p_NtParamCustomerReq				:= ADR(tyNtParamCurr.eCustomerReq);
	p_NtParamProjShutter2Prep			:= ADR(tyNtParamCurr.bProjShutter2Prep);
	p_NtParamProjShutter3Prep			:= ADR(tyNtParamCurr.bProjShutter3Prep);

	//new for Hermes 1.3
	p_NtParamHermesSvyPrep			:= ADR(tyNtParamCurr.bHermesSvyPrep);
	p_NtParamHermesSvyFirstMc		:= ADR(tyNtParamCurr.bHermesSvyFirstMcInTheLine);//First Machine in the line, set for Loader / Destacker
	p_NtParamHermesSvyMagTypeMc		:= ADR(tyNtParamCurr.bHermesSvyMagTypeMc);//Magazine type Machine
	p_NtParamSvyHermesProgNm		:= ADR(tyNtParamCurr.sSvyHermesProgNm);
	p_NtParamSvyHermesConfigFileNm	:= ADR(tyNtParamCurr.sSvyHermesConfigFileNm);
	p_NtParamSvyHermesFileKeepDay	:= ADR(tyNtParamCurr.udiSvyHermesFileKeepDay);
	p_NtParamSvyHermesAliveTmInSec	:= ADR(tyNtParamCurr.udiSvyHermesAliveTmInSec);
	p_NtParamSvyHermesConnTO		:= ADR(tyNtParamCurr.tSvyHermesConnTO);
	p_NtParamSvyHermesRetainFileNm	:= ADR(tyNtParamCurr.sSvyHermesRetainFileNm);
	p_NtParamDSHermesRetainFileNm	:= ADR(tyNtParamCurr.sDSHermesRetainFileNm); //50 Board Data retain file name
	p_NtParamDSHermesMcCycleTm	    := ADR(tyNtParamCurr.rMachineCycleTime); //Machine Board Transfer Cycle Time
	p_NtParamDSHermesAWCycleTm	    := ADR(tyNtParamCurr.rAutoWidthCycleTime); //Machine Autowidth Cycle Time
	p_NtParamHermesScannerPrep    	:= ADR(tyNtParamCurr.bHermesScannerPrep);
	p_NtParamHermesInput            := ADR(tyNtParamCurr.iInput);//Total Input = How many inlet
	p_NtParamHermesOutput           := ADR(tyNtParamCurr.iOutput);//Total Outlet  = How many outlet

	p_NtParamAutoRcpPrep			:= ADR(tyNtParamCurr.bProjAutoRcpPrep);
	p_NtParamAutoRcpParamLmt		:= ADR(tyNtParamCurr.tyAutoRcpParamLmt);
	p_NtParamAutoRcpPrecededBy		:= ADR(tyNtParamCurr.eAutoRcpPrecededBy);

	//Add
	p_NtParmProjChinesePrep				:= ADR(tyNtParamCurr.bchineseprep);
	p_NtParmProjGermanPrep				:= ADR(tyNtParamCurr.bgermanprep);

	p_NtParamProjOutShutter2Prep	:= ADR(tyNtParamCurr.bProjOutShutter2Prep);
	p_NtParamProjCntrPullLmt		:= ADR(tyNtParamCurr.siProjCntrPullLmt);   //pull brd limit
	p_NtParamTrolleyLckPrep			:= ADR(tyNtParamCurr.bProjTrolleyLckPrep);
	p_NtParamTrolleyLckProgNm		:= ADR(tyNtParamCurr.sTrolleyLckProgNm);
	p_NtParamTrolleyLckTwoCtrlIn	:= ADR(tyNtParamCurr.bTrolleyLckTwoCtrlIn);
	p_NtParamTrolleyLckExtTO		:= ADR(tyNtParamCurr.tTrolleyLckExtTO);
	p_NtParamTrolleyLckRetTO		:= ADR(tyNtParamCurr.tTrolleyLckRetTO);

	p_NtParamTrolleyLckProgNm2		:= ADR(tyNtParamCurr.sTrolleyLckProgNm2);
	p_NtParamTrolleyLckTwoCtrlIn2	:= ADR(tyNtParamCurr.bTrolleyLckTwoCtrlIn2);
	p_NtParamTrolleyLckExtTO2		:= ADR(tyNtParamCurr.tTrolleyLckExtTO2);
	p_NtParamTrolleyLckRetTO2		:= ADR(tyNtParamCurr.tTrolleyLckRetTO2);

	(* Always Change If Project Change *)

END_PROGRAM
```

### Program Logical/UsrMgmt/UsrMgmt

#### Act_Alarm.st
```iecst
(** 2019-03-25 **)
ACTION Act_Alarm:

	//Error
	IF EDGEPOS(eStatus = Error) THEN

		tyAlmData.sProgNm		:= p_sProgNm;
		tyAlmData.udiCode		:= udiStatus;
		tyAlmData.eSeverity		:= AlmSeverityError;
		tyAlmData.udiRunTime	:= tyAlmData.udiRunTime + 1;
		tyAlmData.bAlm			:= TRUE;
		tyAlmData.udiModuleNum  := udiModuleNum;
		g_sUsrMgmtProgNm		:= p_sProgNm;
		//Get Error Message
		IF tyAlmData.udiCode < 10000 OR tyAlmData.udiCode > 10099 THEN
			tyAlmData.sAlmMsg	:= 'Unknown';
			tyAlmData.sRcyMsg	:= 'Unknown';
		ELSE
			tyAlmData.sAlmMsg	:= a_tyAlmText[tyAlmData.udiCode].sAlmText;
			tyAlmData.sRcyMsg	:= a_tyAlmText[tyAlmData.udiCode].sRcyText;
		END_IF

		sStatTxt	:= tyAlmData.sAlmMsg;

	ELSIF bRstErr AND (tyAlmData.udiCode <> 0) THEN

		tyAlmData.udiCode	:= 0;
		tyAlmData.eSeverity	:= AlmSeverityNA;
		tyAlmData.sAlmMsg	:= '';
		tyAlmData.sRcyMsg	:= '';
		tyAlmData.bAlm			:= FALSE;
		sStatTxt	:= a_sStatText[eStat];

	END_IF

END_ACTION
```

### Program Logical/Buffer/Buffer1 (IEC) - 1.00.0 - NtBuffer v5.00.0 , NtFileIO v5.00.0

#### InputRef_Link.var
```iecst
(*2019-04-09*)
(**)
(*External*)
VAR
	p_bLinkStartupRun : REFERENCE TO BOOL;
	p_bLinkNtParamProjMagConvPrep : REFERENCE TO BOOL;
	p_eLinkOpsMagLDBufferAct : REFERENCE TO eBufferAction;
	p_eLinkOpsMagConvLDBufferAct : REFERENCE TO eBufferAction;
END_VAR
(**)
VAR
	p_diLinkSltToSltDist : REFERENCE TO DINT;
	p_bLinkMcParamProdSelTopToBtm : REFERENCE TO BOOL;
	p_bLinkPresentSen1 : REFERENCE TO BOOL;
	p_bLinkPresentSen2 : REFERENCE TO BOOL;
END_VAR
(**)
VAR
	p_eLinkMag : REFERENCE TO eLDMag;
	p_usiLinkMod : REFERENCE TO USINT;
END_VAR
(**)
VAR
	p_diLinkMinSlt : REFERENCE TO DINT;
	p_diLinkMaxSlt : REFERENCE TO DINT;
	p_diLinkPitch : REFERENCE TO DINT;
	p_diLinkBffrTtlSlt : REFERENCE TO DINT;
	p_diLinkLifterBtmPosInUM : REFERENCE TO DINT;
END_VAR
(**)
VAR
	p_diLinkSltToSltDist1 : REFERENCE TO DINT;
	p_diLinkMinSlt1 : REFERENCE TO DINT;
	p_diLinkMaxSlt1 : REFERENCE TO DINT;
	p_diLinkPitch1 : REFERENCE TO DINT;
	p_diLinkBffrTtlSlt1 : REFERENCE TO DINT;
	p_diLinkLifterBtmPosInUM1 : REFERENCE TO DINT;
	p_bLinkNtParamProjRotCylPrep : REFERENCE TO BOOL;
END_VAR
(**)
VAR
	p_bLinkProjLifterMagPlatform : REFERENCE TO BOOL;
	p_diNtParamProjMagMaxSlt : REFERENCE TO DINT;
	p_eLinkOpsLifMagLDBufferAct : REFERENCE TO eBufferAction;
	p_bNtParamAutoRcpPrep : REFERENCE TO BOOL;
	p_bMcParamHermesSvyEn : REFERENCE TO BOOL;
	p_bHermesSvyPrep : REFERENCE TO BOOL;
	p_eNtParamCustomerReq : REFERENCE TO eCustomer;
	p_bMcParamMesRFIDEn : REFERENCE TO BOOL;
END_VAR
```

#### Act_InitGlobal.st
```iecst
(** 2019-04-26 **)
ACTION Act_InitGlobal:

	(* Always Change If Project Change *)

	//Pass Data To Link
	p_bLinkStartupRun ACCESS p_StartupRun;
	p_bLinkNtParamProjMagConvPrep ACCESS p_NtParamProjMag1ConvPrep;
//	p_eLinkOpsMagLDBufferAct ACCESS p_OpsMagLD1BufferAct;
	p_eLinkOpsMagConvLDBufferAct ACCESS p_OpsMagConvLD1BufferAct;

	p_bLinkMcParamProdSelTopToBtm ACCESS p_NtParamProjTopToBtmDefault;//p_ProdRcpCurrRcp1TopToBtm;
	p_bLinkPresentSen1 ACCESS p_DIMagPresentSen1;
	p_bLinkPresentSen2 ACCESS p_DIMagConvEntSen1;

	p_eLinkMag ACCESS p_NtParamProjMag;
	p_usiLinkMod ACCESS p_ProdRcpCurrRcp1McMod;

	p_diLinkSltToSltDist ACCESS p_MagRcpCurrRcpSltToSlt;
	p_diLinkMinSlt ACCESS p_ProdRcpCurrRcp1MinSltValue;
	p_diLinkMaxSlt ACCESS p_ProdRcpCurrRcp1MaxSltValue;
	p_diLinkPitch ACCESS p_ProdRcpCurrRcp1Pitch;
	p_diLinkBffrTtlSlt ACCESS p_MagRcpCurrRcpTtlSlt;
	p_diLinkLifterBtmPosInUM ACCESS p_MagRcpCurrRcpMag1Slt1Pos;

	p_diLinkSltToSltDist1 ACCESS p_MagRcpCurrRcpSltToSlt1;
	p_diLinkMinSlt1 ACCESS p_ProdRcpCurrRcp1MinSltRear;
	p_diLinkMaxSlt1 ACCESS p_ProdRcpCurrRcp1MaxSltRear;
	p_diLinkPitch1 ACCESS p_ProdRcpCurrRcp1PitchRear;
	p_diLinkBffrTtlSlt1 ACCESS p_MagRcpCurrRcpTtlSlt1;
	p_diLinkLifterBtmPosInUM1 ACCESS p_MagRcpCurrRcpMag1Slt1Pos1;

	p_bLinkNtParamProjRotCylPrep ACCESS p_NtParamProjPullerRotCylPrep;

	p_bLinkProjLifterMagPlatform ACCESS p_NtParamProjLifterMagPlatform;
	p_diNtParamProjMagMaxSlt ACCESS p_NtParamProjMagMaxSlt; //initial
	p_eLinkOpsLifMagLDBufferAct ACCESS p_OpsLifMagLDBufferAct1;
	p_bNtParamAutoRcpPrep ACCESS p_NtParamAutoRcpPrep;
	p_bHermesSvyPrep ACCESS p_NtParamHermesSvyPrep; //queryWO
	p_bMcParamHermesSvyEn ACCESS p_McParamHermesSvyEn;
	p_eNtParamCustomerReq ACCESS p_NtParamCustomerReq;
	p_bMcParamMesRFIDEn ACCESS p_McParamMesRFIDEn;

	//Pass Data To Internal Use
	p_udiRstErr ACCESS p_RstErrReset;
	p_sFileName ACCESS p_NtParamBffr1FileNm;
	p_bManual ACCESS p_UIMnlMod;
	p_dtCurrDT ACCESS p_TimeCurrDT;
//	p_diMinSlt ACCESS p_ProdRcpCurrRcp1MinSltValue;
//	p_diMaxSlt ACCESS p_ProdRcpCurrRcp1MaxSltValue;
//	p_diPitch ACCESS p_ProdRcpCurrRcp1Pitch;
//	p_diBffrTtlSlt ACCESS p_MagRcpCurrRcpTtlSlt;
//	p_diLifterBtmPosInUM ACCESS p_MagRcpCurrRcpMag1Slt1Pos;
	p_diLifterCurrPosInUM ACCESS p_LifterBtmActualPos;
	p_bFIFO ACCESS p_NtParamBffr1FIFO;
//	p_bMagPresentSensor ACCESS p_DIMagPresentSen1;
	p_sCurrRcpNm ACCESS p_ProdRcpCurrRcp1Nm;
	p_sProgNm ACCESS p_NtParamBffr1ProgNm;
	p_bNtSettingsLoadDone ACCESS p_StartupNtSettingsLoadDone;

	(* Always Change If Project Change *)

END_ACTION
```

#### Act_Initial.st
```iecst
(** 2019-04-26 **)
ACTION Act_Initial:

	//Initial
	sStatTxt	:= a_sStatText[eStat];

	fbDirCreate1.sDevice	:= 'F';
	fbDirCreate1.sDirName	:= 'User';
	fbDirCreate1(bEn := FALSE);

	fbDirCreate2.sDevice	:= 'User';
	fbDirCreate2.sDirName	:= 'Retain';
	fbDirCreate2(bEn := FALSE);

	fbFileRead1.sDevice			:= 'Retain';
	fbFileRead1.sFile			:= p_sFileName;
	fbFileRead1.udiOffset		:= 0;
	fbFileRead1.p_Dest			:= ADR(p_tyBuffer);
	fbFileRead1.udiLen			:= SIZEOF(p_tyBuffer);
	fbFileRead1(bEn := FALSE);

	fbFileWrite1.sDevice		:= 'Retain';
	fbFileWrite1.sFile			:= p_sFileName;
	fbFileWrite1.udiOffset		:= 0;
	fbFileWrite1.p_Src			:= ADR(p_tyBuffer);
	fbFileWrite1.udiLen			:= SIZEOF(p_tyBuffer);
	fbFileWrite1.udiOption		:= 0;
	fbFileWrite1(bEn := FALSE);

	fbCoolFanOffDlyTm.PT	:= DINT_TO_TIME(p_diCoolFanOffDlyTm);
	fbCoolFanOffDlyTm(IN := FALSE);

	fbCoolFanOffChkTm(IN := FALSE);
	fbMagAbsentTm(IN := FALSE);
	fbMagPresentTm(IN := FALSE);

	IF p_bLinkMcParamProdSelTopToBtm THEN
		diNxtUnloadSlt := 0;
	ELSE
		diNxtUnloadSlt := p_diNtParamProjMagMaxSlt;
	END_IF

END_ACTION
```

#### Act_Link.st
```iecst
(** 2019-03-29 **)
ACTION Act_Link:

	IF p_eLinkMag = LDMagQuadruple THEN
		CASE p_usiLinkMod OF
			0,2:  //LDModLoadLnA, LDModLoadLnAB:
				IF p_bAscending THEN
					p_diSltToSltInUM := p_diLinkSltToSltDist * -1;
				ELSE
					p_diSltToSltInUM := p_diLinkSltToSltDist;
				END_IF
				p_diMinSlt := p_diLinkMinSlt;
				p_diMaxSlt := p_diLinkMaxSlt;
				p_diPitch := p_diLinkPitch;
				p_diBffrTtlSlt := p_diLinkBffrTtlSlt;
				p_diLifterBtmPosInUM := p_diLinkLifterBtmPosInUM;

			1: //LDModLoadLnB:
				IF p_bAscending THEN
					p_diSltToSltInUM := p_diLinkSltToSltDist1 * -1;
				ELSE
					p_diSltToSltInUM := p_diLinkSltToSltDist1;
				END_IF
				p_diSltToSltInUM := p_diLinkSltToSltDist1;
				p_diMinSlt := p_diLinkMinSlt1;
				p_diMaxSlt := p_diLinkMaxSlt1;
				p_diPitch := p_diLinkPitch1;
				p_diBffrTtlSlt := p_diLinkBffrTtlSlt1;
				p_diLifterBtmPosInUM := p_diLinkLifterBtmPosInUM1;

		END_CASE
	ELSE

		IF p_bAscending THEN
			p_diSltToSltInUM := p_diLinkSltToSltDist * -1;
		ELSE
			p_diSltToSltInUM := p_diLinkSltToSltDist;
		END_IF
		IF p_bNtParamAutoRcpPrep AND ((p_bHermesSvyPrep AND p_bMcParamHermesSvyEn) OR (p_eNtParamCustomerReq = We_Fabricate AND p_bMcParamMesRFIDEn)) THEN
			p_diMinSlt ACCESS p_diAutoRcpMag1MinSlt;
			p_diMaxSlt ACCESS p_diAutoRcpMag1MaxSlt;
			p_diPitch ACCESS p_diAutoRcpMag1Pitch;
		ELSE
			p_diMinSlt ACCESS ADR(diMinSlt);
			p_diMaxSlt ACCESS ADR(diMaxSlt);
			p_diPitch ACCESS ADR(diPitch);
			p_diMinSlt := p_diLinkMinSlt;
			p_diMaxSlt := p_diLinkMaxSlt;
			p_diPitch := p_diLinkPitch;
		END_IF
		p_diBffrTtlSlt := p_diLinkBffrTtlSlt;
		p_diLifterBtmPosInUM := p_diLinkLifterBtmPosInUM;
	END_IF

	p_bAscending	:= NOT p_bLinkMcParamProdSelTopToBtm;
//	IF p_bLinkNtParamProjRotCylPrep THEN
//		p_bAscending := TRUE;
//	ELSE
//		p_bAscending := FALSE;
//	END_IF

	IF p_bLinkNtParamProjMagConvPrep THEN
		fbMagPresentTm.PT	:= T#2s;
	ELSE
		fbMagPresentTm.PT	:= T#8s;
	END_IF

	p_bMagPresentSensor := p_bLinkPresentSen1 OR p_bLinkPresentSen2;

END_ACTION
```

#### Act_LinkAction.st
```iecst
(** 2019-05-10 **)
ACTION Act_LinkAction:

	IF p_bLinkStartupRun = TRUE THEN
		p_eAct ACCESS p_StartupBuffer1Act;
	ELSE
		IF eStatus = Idle THEN
			IF p_bLinkProjLifterMagPlatform = FALSE THEN
				IF p_eLinkOpsMagConvLDBufferAct <> BufferActIdle THEN
					p_eAct ACCESS p_OpsMagConvLD1BufferAct;
				ELSE
					p_eAct ACCESS p_UIBuffer1Act;
				END_IF
			ELSE
				IF p_eLinkOpsLifMagLDBufferAct <> BufferActIdle THEN
					p_eAct ACCESS p_OpsLifMagLDBufferAct1;
				ELSE
					p_eAct ACCESS p_UIBuffer1Act;
				END_IF
			END_IF
		END_IF
	END_IF

END_ACTION
```

#### Act_Main.st
```iecst
(** 2019-07-03 **)
ACTION Act_Main:

	IF eStatOld <> eStat THEN
		fbDirCreate1(bEn := FALSE);
		fbDirCreate2(bEn := FALSE);
		fbFileRead1(bEn := FALSE);
		fbFileWrite1(bEn := FALSE);
		usiStep	:= 0;

		bFileNotFound			:= FALSE;
		bNewProduct				:= FALSE;
		bLastProductUnload		:= FALSE;
		bLastProductLeftInBffr	:= FALSE;

		sStatTxt	:= a_sStatText[eStat];

		eStatOld	:= eStat;

		eStatus		:= Busy;
	END_IF

	//Main
	CASE eStat OF

		BufferActIdle:
			eStatus	:= Idle;

		BufferActCreateDir:
			IF eStatus = Idle OR eStatus = Busy THEN

				eStatus	:= Busy;

				CASE usiStep OF
					0:
						fbDirCreate1(bEn := TRUE);
						IF fbDirCreate1.udiStatus = 0 THEN
							usiStep	:= 1;
						ELSIF fbDirCreate1.udiStatus < 65534 THEN
							eStatus		:= Error;

							IF fbDirCreate1.udiStatus = 1908 THEN
								udiStatus	:= 10000;	//Create User Directory Error
							ELSE
								udiStatus	:= fbDirCreate1.udiStatus;
							END_IF
						END_IF

					1:
						fbDirCreate2(bEn := TRUE);
						IF fbDirCreate2.udiStatus = 0 THEN
							eStatus	:= Done;
						ELSIF fbDirCreate2.udiStatus < 65534 THEN
							eStatus		:= Error;

							IF fbDirCreate2.udiStatus = 1908 THEN
								udiStatus	:= 10001;	//Create Retain Directory Error
							ELSE
								udiStatus	:= fbDirCreate2.udiStatus;
							END_IF
						END_IF

				END_CASE

			END_IF

		BufferActGetRetainBffr:
			IF eStatus = Idle OR eStatus = Busy THEN

				eStatus	:= Busy;

				fbFileRead1(bEn := TRUE);
				IF fbFileRead1.udiStatus = 0 THEN
					eStatus	:= Done;

					tyBffrParameter.diBffrTtlSlt	:= p_diBffrTtlSlt;
					tyBffrParameter.diSltCap		:= p_diSltCap;

					fBffrStat(ADR(p_tyBufferStat) , p_tyBuffer);
					fDispBffrDescending(ADR(p_tyDispBuffer) , tyBffrParameter , p_tyBuffer , p_dtCurrDT , DINT_TO_TIME(p_diCoolTm) , 0 , 1 , 2);

				ELSIF fbFileRead1.udiStatus < 65534 THEN
					eStatus	:= Error;

					IF fbFileRead1.udiStatus = 1900 THEN
						udiStatus	:= 10002;	//File Open Error While Reading Retain File
					ELSIF fbFileRead1.udiStatus = 1902 THEN
						udiStatus	:= 10003;	//File Read Error While Reading Retain File
					ELSIF fbFileRead1.udiStatus = 1904 THEN
						udiStatus	:= 10004;	//File Close Error While Reading Retain File
					ELSIF fbFileRead1.udiStatus = 1915 THEN
						eStatus			:= Done;
						bFileNotFound	:= TRUE;
					ELSE
						udiStatus	:= fbFileRead1.udiStatus;
					END_IF
				END_IF

			END_IF

		BufferActSetFull:
			IF eStatus = Idle OR eStatus = Busy THEN

				eStatus	:= Busy;

				CASE usiStep OF
					0:
						tyBffrParameter.bAscending		:= p_bAscending;
						tyBffrParameter.diBffrTtlSlt	:= p_diBffrTtlSlt;
						tyBffrParameter.diMaxSlt		:= p_diMaxSlt;
						tyBffrParameter.diMinSlt		:= p_diMinSlt;
						tyBffrParameter.diPitch			:= p_diPitch;
						tyBffrParameter.diSltCap		:= p_diSltCap;
						tyBffrParameter.a_bSkip			:= pa_bSkip;
						bFIFOOld						:= p_bFIFO;

						udiStatus	:= fBffrSetFull(ADR(p_tyBuffer) , tyBffrParameter , p_dtCurrDT , p_sBffrNm , p_sProdNm);

						IF udiStatus = 0 THEN
							usiStep	:= 1;

							fBffrStat(ADR(p_tyBufferStat) , p_tyBuffer);
							fDispBffrDescending(ADR(p_tyDispBuffer) , tyBffrParameter , p_tyBuffer , p_dtCurrDT , DINT_TO_TIME(p_diCoolTm) , 0 , 1 , 2);

						ELSE
							eStatus	:= Error;

						END_IF

					1:
						fbFileWrite1(bEn := TRUE);

						IF fbFileWrite1.udiStatus = 0 THEN
							eStatus	:= Done;
						ELSIF fbFileWrite1.udiStatus < 65534 THEN
							eStatus	:= Error;

							IF fbFileWrite1.udiStatus = 1900 THEN
								udiStatus	:= 10005;	//File Open Error While Setting Full Buffer
							ELSIF fbFileWrite1.udiStatus = 1901 THEN
								udiStatus	:= 10006;	//File Create Error While Setting Full Buffer
							ELSIF fbFileWrite1.udiStatus = 1903 THEN
								udiStatus	:= 10007;	//File Write Error While Setting Full Buffer
							ELSIF fbFileWrite1.udiStatus = 1904 THEN
								udiStatus	:= 10008;	//File Close Error While Setting Full Buffer
							ELSIF fbFileWrite1.udiStatus = 1914 THEN
								udiStatus	:= 10040;	//Directory Does Not Exist While Setting Full Buffer
							ELSE
								udiStatus	:= fbFileWrite1.udiStatus;
							END_IF
						END_IF

				END_CASE

			END_IF

		BufferActSetMty:
			IF eStatus = Idle OR eStatus = Busy THEN

				eStatus	:= Busy;

				CASE usiStep OF
					0:
						tyBffrParameter.bAscending		:= p_bAscending;
						tyBffrParameter.diBffrTtlSlt	:= p_diBffrTtlSlt;
						tyBffrParameter.diMaxSlt		:= p_diMaxSlt;
						tyBffrParameter.diMinSlt		:= p_diMinSlt;
						tyBffrParameter.diPitch			:= p_diPitch;
						tyBffrParameter.diSltCap		:= p_diSltCap;
						tyBffrParameter.a_bSkip			:= pa_bSkip;
						bFIFOOld						:= p_bFIFO;

						udiStatus	:= fBffrSetMty(ADR(p_tyBuffer) , tyBffrParameter , p_sBffrNm);

						IF udiStatus = 0 THEN
							usiStep	:= 1;

							fBffrStat(ADR(p_tyBufferStat) , p_tyBuffer);
							fDispBffrDescending(ADR(p_tyDispBuffer) , tyBffrParameter , p_tyBuffer , p_dtCurrDT , DINT_TO_TIME(p_diCoolTm) , 0 , 1 , 2);

						ELSE
							eStatus	:= Error;

						END_IF

					1:
						fbFileWrite1(bEn := TRUE);

						IF fbFileWrite1.udiStatus = 0 THEN
							eStatus	:= Done;
						ELSIF fbFileWrite1.udiStatus < 65534 THEN
							eStatus	:= Error;

							IF fbFileWrite1.udiStatus = 1900 THEN
								udiStatus	:= 10009;	//File Open Error While Setting Empty Buffer
							ELSIF fbFileWrite1.udiStatus = 1901 THEN
								udiStatus	:= 10010;	//File Create Error While Setting Empty Buffer
							ELSIF fbFileWrite1.udiStatus = 1903 THEN
								udiStatus	:= 10011;	//File Write Error While Setting Empty Buffer
							ELSIF fbFileWrite1.udiStatus = 1904 THEN
								udiStatus	:= 10012;	//File Close Error While Setting Empty Buffer
							ELSIF fbFileWrite1.udiStatus = 1914 THEN
								udiStatus	:= 10041;	//Directory Does Not Exist While Setting Empty Buffer
							ELSE
								udiStatus	:= fbFileWrite1.udiStatus;
							END_IF
						END_IF

				END_CASE

			END_IF

		BufferActLoad:
			IF eStatus = Idle OR eStatus = Busy THEN

				eStatus	:= Busy;

				CASE usiStep OF
					0:
						diCurrSlt	:= fLifterPosInUMToSltBtmMin(p_diLifterCurrPosInUM , p_diSltToSltInUM , p_diLifterBtmPosInUM);

						udiStatus	:= fBffrLoad(ADR(p_tyBuffer) , ADR(bNewProduct) , diCurrSlt , p_dtCurrDT , p_bGdBrdIn , p_sProdNm , p_sBarcode1 , p_sBarcode2);

						IF udiStatus = 0 THEN
							usiStep	:= 1;

							tyBffrParameter.diBffrTtlSlt	:= p_diBffrTtlSlt;
							tyBffrParameter.diSltCap		:= p_diSltCap;

							fBffrStat(ADR(p_tyBufferStat) , p_tyBuffer);
							fDispBffrDescending(ADR(p_tyDispBuffer) , tyBffrParameter , p_tyBuffer , p_dtCurrDT , DINT_TO_TIME(p_diCoolTm) , 0 , 1 , 2);

						ELSE
							eStatus	:= Error;

							IF udiStatus = 1010 THEN
								udiStatus	:= 10076;	//Loading Slot Is Not For Board
							ELSIF udiStatus = 1011 THEN
								udiStatus	:= 10077;	//Loading Slot Is Full Of Board
							ELSIF udiStatus = 1012 THEN
								udiStatus	:= 10078;	//Loading First Sub-Slot Is Not For Board
							ELSIF udiStatus	= 1013 THEN
								udiStatus	:= 10079;	//Loading Last Sub-Slot Have Board, Which Mean Slot Is Full Of Board
							ELSIF udiStatus = 1014 THEN
								udiStatus	:= 10080;	//Loading Last Sub-Slot Is Not For Board
							ELSIF udiStatus = 1015 THEN
								udiStatus	:= 10081;	//Loading Slot Is Full Of Board
							ELSIF udiStatus = 1001 THEN
								udiStatus	:= 10082;	//Loading Slot Is Skipped
							ELSIF udiStatus	= 1016 THEN
								udiStatus	:= 10083;	//Existing Board Status Is Different With Loading Board Status
							END_IF

						END_IF

					1:
						fbFileWrite1(bEn := TRUE);

						IF fbFileWrite1.udiStatus = 0 THEN
							eStatus	:= Done;
						ELSIF fbFileWrite1.udiStatus < 65534 THEN
							eStatus	:= Error;

							IF fbFileWrite1.udiStatus = 1900 THEN
								udiStatus	:= 10013;	//File Open Error While Loading Info To Buffer
							ELSIF fbFileWrite1.udiStatus = 1901 THEN
								udiStatus	:= 10014;	//File Create Error While Loading Info To Buffer
							ELSIF fbFileWrite1.udiStatus = 1903 THEN
								udiStatus	:= 10015;	//File Write Error While Loading Info To Buffer
							ELSIF fbFileWrite1.udiStatus = 1904 THEN
								udiStatus	:= 10016;	//File Close Error While Loading Info To Buffer
							ELSIF fbFileWrite1.udiStatus = 1914 THEN
								udiStatus	:= 10042;	//Directory Does Not Exist While Loading Info To Buffer
							ELSE
								udiStatus	:= fbFileWrite1.udiStatus;
							END_IF
						END_IF

				END_CASE

			END_IF

		BufferActLoadSltChk:
			IF eStatus = Idle OR eStatus = Busy THEN

				eStatus	:= Busy;

				CASE usiStep OF
					0:
						diCurrSlt	:= fLifterPosInUMToSltBtmMin(p_diLifterCurrPosInUM , p_diSltToSltInUM , p_diLifterBtmPosInUM);

						IF p_bNxtLoadSeq = TRUE AND p_bGdBrdIn = TRUE THEN
							diExpectedSlt	:= fBffrNxtLoadSeqGd(p_bAscending , p_tyBuffer);
						ELSIF p_bNxtLoadSeq = TRUE AND p_bGdBrdIn = FALSE THEN
							diExpectedSlt	:= fBffrNxtLoadSeqBad(p_bAscending , p_tyBuffer);
						ELSIF p_bNxtLoadSeq = FALSE AND p_bGdBrdIn = TRUE THEN
							diExpectedSlt	:= fBffrNxtLoadNearbyGd(diCurrSlt , p_tyBuffer);
						ELSE
							diExpectedSlt	:= fBffrNxtLoadNearbyBad(diCurrSlt , p_tyBuffer);
						END_IF

						IF diCurrSlt = diExpectedSlt THEN
							udiStatus	:= fBffrLoad(ADR(p_tyBuffer) , ADR(bNewProduct) , diCurrSlt , p_dtCurrDT , p_bGdBrdIn , p_sProdNm , p_sBarcode1 , p_sBarcode2);

							IF udiStatus = 0 THEN
								usiStep	:= 1;

								tyBffrParameter.diBffrTtlSlt	:= p_diBffrTtlSlt;
								tyBffrParameter.diSltCap		:= p_diSltCap;

								fBffrStat(ADR(p_tyBufferStat) , p_tyBuffer);
								fDispBffrDescending(ADR(p_tyDispBuffer) , tyBffrParameter , p_tyBuffer , p_dtCurrDT , DINT_TO_TIME(p_diCoolTm) , 0 , 1 , 2);

							ELSE
								eStatus	:= Error;

								IF udiStatus = 1010 THEN
									udiStatus	:= 10084;	//Loading Slot Is Not For Board
								ELSIF udiStatus = 1011 THEN
									udiStatus	:= 10085;	//Loading Slot Is Full Of Board
								ELSIF udiStatus = 1012 THEN
									udiStatus	:= 10086;	//Loading First Sub-Slot Is Not For Board
								ELSIF udiStatus	= 1013 THEN
									udiStatus	:= 10087;	//Loading Last Sub-Slot Have Board, Which Mean Slot Is Full Of Board
								ELSIF udiStatus = 1014 THEN
									udiStatus	:= 10088;	//Loading Last Sub-Slot Is Not For Board
								ELSIF udiStatus = 1015 THEN
									udiStatus	:= 10089;	//Loading Slot Is Full Of Board
								ELSIF udiStatus = 1001 THEN
									udiStatus	:= 10090;	//Loading Slot Is Skipped
								ELSIF udiStatus	= 1016 THEN
									udiStatus	:= 10091;	//Existing Board Status Is Different With Loading Board Status
								END_IF

							END_IF

						ELSE
							udiStatus	:= 10017;	//Wrong Slot Number To Load
							eStatus		:= Error;

						END_IF

					1:
						fbFileWrite1(bEn := TRUE);

						IF fbFileWrite1.udiStatus = 0 THEN
							eStatus	:= Done;
						ELSIF fbFileWrite1.udiStatus < 65534 THEN
							eStatus	:= Error;

							IF fbFileWrite1.udiStatus = 1900 THEN
								udiStatus	:= 10018;	//File Open Error While Loading Info To Buffer With Slot Check
							ELSIF fbFileWrite1.udiStatus = 1901 THEN
								udiStatus	:= 10019;	//File Create Error While Loading Info To Buffer With Slot Check
							ELSIF fbFileWrite1.udiStatus = 1903 THEN
								udiStatus	:= 10020;	//File Write Error While Loading Info To Buffer With Slot Check
							ELSIF fbFileWrite1.udiStatus = 1904 THEN
								udiStatus	:= 10021;	//File Close Error While Loading Info To Buffer With Slot Check
							ELSIF fbFileWrite1.udiStatus = 1914 THEN
								udiStatus	:= 10043;	//Directory Does Not Exist While Loading Info To Buffer With Slot Check
							ELSE
								udiStatus	:= fbFileWrite1.udiStatus;
							END_IF
						END_IF

				END_CASE

			END_IF

		BufferActUnload:
			IF eStatus = Idle OR eStatus = Busy THEN

				eStatus	:= Busy;

				CASE usiStep OF
					0:
						IF p_bLinkMcParamProdSelTopToBtm AND p_bLinkProjLifterMagPlatform = FALSE THEN //TravLif with fixed puller
							diCurrSlt	:= fLifterPosInUMToSltTopMin(p_diLifterCurrPosInUM , p_diSltToSltInUM , p_diLifterBtmPosInUM); //Slt to slt positive
						ELSE
							diCurrSlt	:= fLifterPosInUMToSltBtmMin(p_diLifterCurrPosInUM , p_diSltToSltInUM , p_diLifterBtmPosInUM);
						END_IF

						udiStatus	:= fBffrUnload(ADR(tyBoardUnloadStat) , ADR(p_tyBuffer) , ADR(bLastProductUnload) , ADR(bLastProductLeftInBffr) , diCurrSlt);

						IF p_sCurrRcpNm = tyBoardUnloadStat.sProdNm THEN
							bLastProductUnload	:= FALSE;
						END_IF

						IF udiStatus = 0 THEN
							usiStep	:= 1;

							tyBffrParameter.diBffrTtlSlt	:= p_diBffrTtlSlt;
							tyBffrParameter.diSltCap		:= p_diSltCap;

							fBffrStat(ADR(p_tyBufferStat) , p_tyBuffer);
							fDispBffrDescending(ADR(p_tyDispBuffer) , tyBffrParameter , p_tyBuffer , p_dtCurrDT , DINT_TO_TIME(p_diCoolTm) , 0 , 1 , 2);

						ELSE
							eStatus	:= Error;

							IF udiStatus = 1000 THEN
								udiStatus	:= 10048;	//Unloading Slot Is Skipped While Unloading Buffer
							ELSIF udiStatus = 1003 THEN
								udiStatus	:= 10049;	//Unloading Slot Is Not For Board While Unloading Buffer
							ELSIF udiStatus = 1004 THEN
								udiStatus	:= 10050;	//Unloading Slot Board Is Not available While Unloading Buffer
							ELSIF udiStatus = 1005 THEN
								udiStatus	:= 10051;	//Unloading Last Sub Slot Is Not For Board While Unloading Buffer
							ELSIF udiStatus = 1006 THEN
								udiStatus	:= 10052;	//Unloading Last Sub Slot Has No Board While Unloading Buffer
							ELSIF udiStatus = 1007 THEN
								udiStatus	:= 10053;	//Board Quantity In Slot Is 0 While Unloading Buffer
							ELSIF udiStatus = 1008 THEN
								udiStatus	:= 10054;	//Board Capacity In Slot Is 0 While Unloading Buffer
							END_IF

						END_IF

					1:
						fbFileWrite1(bEn := TRUE);

						IF fbFileWrite1.udiStatus = 0 THEN
							eStatus	:= Done;
						ELSIF fbFileWrite1.udiStatus < 65534 THEN
							eStatus	:= Error;

							IF fbFileWrite1.udiStatus = 1900 THEN
								udiStatus	:= 10022;	//File Open Error While Unloading Info From Buffer
							ELSIF fbFileWrite1.udiStatus = 1901 THEN
								udiStatus	:= 10023;	//File Create Error While Unloading Info From Buffer
							ELSIF fbFileWrite1.udiStatus = 1903 THEN
								udiStatus	:= 10024;	//File Write Error While Unloading Info From Buffer
							ELSIF fbFileWrite1.udiStatus = 1904 THEN
								udiStatus	:= 10025;	//File Close Error While Unloading Info From Buffer
							ELSIF fbFileWrite1.udiStatus = 1914 THEN
								udiStatus	:= 10044;	//Directory Does Not Exist While Unloading Info From Buffer
							ELSE
								udiStatus	:= fbFileWrite1.udiStatus;
							END_IF
						END_IF

				END_CASE

			END_IF

		BufferActUnloadSltChk:
			IF eStatus = Idle OR eStatus = Busy THEN

				eStatus	:= Busy;

				CASE usiStep OF
					0:
						diCurrSlt	:= fLifterPosInUMToSltBtmMin(p_diLifterCurrPosInUM , p_diSltToSltInUM , p_diLifterBtmPosInUM);

						IF p_bFIFO = TRUE AND p_bGdBrdReq = TRUE THEN
							diExpectedSlt	:= fBffrNxtUnloadFIFOGd(p_tyBuffer , '');
						ELSIF p_bFIFO = TRUE AND p_bGdBrdReq = FALSE THEN
							diExpectedSlt	:= fBffrNxtUnloadFIFOBad(p_tyBuffer , '');
						ELSIF p_bFIFO = FALSE AND p_bGdBrdReq = TRUE THEN
							diExpectedSlt	:= fBffrNxtUnloadLIFOGd(p_tyBuffer , '');
						ELSE
							diExpectedSlt	:= fBffrNxtUnloadLIFOBad(p_tyBuffer , '');
						END_IF

						IF diCurrSlt = diExpectedSlt THEN
							udiStatus	:= fBffrUnload(ADR(tyBoardUnloadStat) , ADR(p_tyBuffer) , ADR(bLastProductUnload) , ADR(bLastProductLeftInBffr) , diCurrSlt);

							IF p_sCurrRcpNm = tyBoardUnloadStat.sProdNm THEN
								bLastProductUnload	:= FALSE;
							END_IF

							IF udiStatus = 0 THEN
								usiStep	:= 1;

								tyBffrParameter.diBffrTtlSlt	:= p_diBffrTtlSlt;
								tyBffrParameter.diSltCap		:= p_diSltCap;

								fBffrStat(ADR(p_tyBufferStat) , p_tyBuffer);
								fDispBffrDescending(ADR(p_tyDispBuffer) , tyBffrParameter , p_tyBuffer , p_dtCurrDT , DINT_TO_TIME(p_diCoolTm) , 0 , 1 , 2);

							ELSE
								eStatus	:= Error;

								IF udiStatus = 1000 THEN
									udiStatus	:= 10055;	//Unloading Slot Is Skipped While Unloading Buffer With Slot Check
								ELSIF udiStatus = 1003 THEN
									udiStatus	:= 10056;	//Unloading Slot Is Not For Board While Unloading Buffer With Slot Check
								ELSIF udiStatus = 1004 THEN
									udiStatus	:= 10057;	//Unloading Slot Board Is Not available While Unloading Buffer With Slot Check
								ELSIF udiStatus = 1005 THEN
									udiStatus	:= 10058;	//Unloading Last Sub Slot Is Not For Board While Unloading Buffer With Slot Check
								ELSIF udiStatus = 1006 THEN
									udiStatus	:= 10059;	//Unloading Last Sub Slot Has No Board While Unloading Buffer With Slot Check
								ELSIF udiStatus = 1007 THEN
									udiStatus	:= 10060;	//Board Quantity In Slot Is 0 While Unloading Buffer With Slot Check
								ELSIF udiStatus = 1008 THEN
									udiStatus	:= 10061;	//Board Capacity In Slot Is 0 While Unloading Buffer With Slot Check
								END_IF

							END_IF

						ELSE
							udiStatus	:= 10026;	//Wrong Slot Number To Unload
							eStatus		:= Error;

						END_IF

					1:
						fbFileWrite1(bEn := TRUE);

						IF fbFileWrite1.udiStatus = 0 THEN
							eStatus	:= Done;
						ELSIF fbFileWrite1.udiStatus < 65534 THEN
							eStatus	:= Error;

							IF fbFileWrite1.udiStatus = 1900 THEN
								udiStatus	:= 10027;	//File Open Error While Unloading Info From Buffer With Slot Check
							ELSIF fbFileWrite1.udiStatus = 1901 THEN
								udiStatus	:= 10028;	//File Create Error While Unloading Info From Buffer With Slot Check
							ELSIF fbFileWrite1.udiStatus = 1903 THEN
								udiStatus	:= 10029;	//File Write Error While Unloading Info From Buffer With Slot Check
							ELSIF fbFileWrite1.udiStatus = 1904 THEN
								udiStatus	:= 10030;	//File Close Error While Unloading Info From Buffer With Slot Check
							ELSIF fbFileWrite1.udiStatus = 1914 THEN
								udiStatus	:= 10045;	//Directory Does Not Exist While Unloading Info From Buffer With Slot Check
							ELSE
								udiStatus	:= fbFileWrite1.udiStatus;
							END_IF
						END_IF

				END_CASE

			END_IF

		BufferActUnloadCoolChk:
			IF eStatus = Idle OR eStatus = Busy THEN

				eStatus	:= Busy;

				CASE usiStep OF
					0:
						diCurrSlt	:= fLifterPosInUMToSltBtmMin(p_diLifterCurrPosInUM , p_diSltToSltInUM , p_diLifterBtmPosInUM);

						bCoolNotRdy	:= NOT fBffrChkCoolTmRdy(diCurrSlt, p_dtCurrDT, DINT_TO_TIME(p_diCoolTm), p_tyBuffer);

						IF bCoolNotRdy = FALSE THEN
							udiStatus	:= fBffrUnload(ADR(tyBoardUnloadStat) , ADR(p_tyBuffer) , ADR(bLastProductUnload) , ADR(bLastProductLeftInBffr) , diCurrSlt);

							IF p_sCurrRcpNm = tyBoardUnloadStat.sProdNm THEN
								bLastProductUnload	:= FALSE;
							END_IF

							IF udiStatus = 0 THEN
								usiStep	:= 1;

								tyBffrParameter.diBffrTtlSlt	:= p_diBffrTtlSlt;
								tyBffrParameter.diSltCap		:= p_diSltCap;

								fBffrStat(ADR(p_tyBufferStat) , p_tyBuffer);
								fDispBffrDescending(ADR(p_tyDispBuffer) , tyBffrParameter , p_tyBuffer , p_dtCurrDT , DINT_TO_TIME(p_diCoolTm) , 0 , 1 , 2);

							ELSE
								eStatus	:= Error;

								IF udiStatus = 1000 THEN
									udiStatus	:= 10062;	//Unloading Slot Is Skipped While Unloading Buffer With Cool Check
								ELSIF udiStatus = 1003 THEN
									udiStatus	:= 10063;	//Unloading Slot Is Not For Board While Unloading Buffer With Cool Check
								ELSIF udiStatus = 1004 THEN
									udiStatus	:= 10064;	//Unloading Slot Board Is Not available While Unloading Buffer With Cool Check
								ELSIF udiStatus = 1005 THEN
									udiStatus	:= 10065;	//Unloading Last Sub Slot Is Not For Board While Unloading Buffer With Cool Check
								ELSIF udiStatus = 1006 THEN
									udiStatus	:= 10066;	//Unloading Last Sub Slot Has No Board While Unloading Buffer With Cool Check
								ELSIF udiStatus = 1007 THEN
									udiStatus	:= 10067;	//Board Quantity In Slot Is 0 While Unloading Buffer With Cool Check
								ELSIF udiStatus = 1008 THEN
									udiStatus	:= 10068;	//Board Capacity In Slot Is 0 While Unloading Buffer With Cool Check
								END_IF

							END_IF

						ELSE
							eStatus	:= Done;

						END_IF

					1:
						fbFileWrite1(bEn := TRUE);

						IF fbFileWrite1.udiStatus = 0 THEN
							eStatus	:= Done;
						ELSIF fbFileWrite1.udiStatus < 65534 THEN
							eStatus	:= Error;

							IF fbFileWrite1.udiStatus = 1900 THEN
								udiStatus	:= 10031;	//File Open Error While Unloading Info From Buffer With Cooling Time Check
							ELSIF fbFileWrite1.udiStatus = 1901 THEN
								udiStatus	:= 10032;	//File Create Error While Unloading Info From Buffer With Cooling Time Check
							ELSIF fbFileWrite1.udiStatus = 1903 THEN
								udiStatus	:= 10033;	//File Write Error While Unloading Info From Buffer With Cooling Time Check
							ELSIF fbFileWrite1.udiStatus = 1904 THEN
								udiStatus	:= 10034;	//File Close Error While Unloading Info From Buffer With Cooling Time Check
							ELSIF fbFileWrite1.udiStatus = 1914 THEN
								udiStatus	:= 10046;	//Directory Does Not Exist While Unloading Info From Buffer With Cooling Time Check
							ELSE
								udiStatus	:= fbFileWrite1.udiStatus;
							END_IF
						END_IF

				END_CASE

			END_IF

		BufferActUnloadSltChkCoolChk:
			IF eStatus = Idle OR eStatus = Busy THEN

				eStatus	:= Busy;

				CASE usiStep OF
					0:
						diCurrSlt	:= fLifterPosInUMToSltBtmMin(p_diLifterCurrPosInUM , p_diSltToSltInUM , p_diLifterBtmPosInUM);

						IF p_bFIFO = TRUE AND p_bGdBrdReq = TRUE THEN
							diExpectedSlt	:= fBffrNxtUnloadFIFOGd(p_tyBuffer , '');
						ELSIF p_bFIFO = TRUE AND p_bGdBrdReq = FALSE THEN
							diExpectedSlt	:= fBffrNxtUnloadFIFOBad(p_tyBuffer , '');
						ELSIF p_bFIFO = FALSE AND p_bGdBrdReq = TRUE THEN
							diExpectedSlt	:= fBffrNxtUnloadLIFOGd(p_tyBuffer , '');
						ELSE
							diExpectedSlt	:= fBffrNxtUnloadLIFOBad(p_tyBuffer , '');
						END_IF

						IF diCurrSlt = diExpectedSlt THEN
							bCoolNotRdy	:= NOT fBffrChkCoolTmRdy(diCurrSlt, p_dtCurrDT, DINT_TO_TIME(p_diCoolTm), p_tyBuffer);

							IF bCoolNotRdy = FALSE THEN
								udiStatus	:= fBffrUnload(ADR(tyBoardUnloadStat) , ADR(p_tyBuffer) , ADR(bLastProductUnload) , ADR(bLastProductLeftInBffr) , diCurrSlt);

								IF p_sCurrRcpNm = tyBoardUnloadStat.sProdNm THEN
									bLastProductUnload	:= FALSE;
								END_IF

								IF udiStatus = 0 THEN
									usiStep	:= 1;

									tyBffrParameter.diBffrTtlSlt	:= p_diBffrTtlSlt;
									tyBffrParameter.diSltCap		:= p_diSltCap;

									fBffrStat(ADR(p_tyBufferStat) , p_tyBuffer);
									fDispBffrDescending(ADR(p_tyDispBuffer) , tyBffrParameter , p_tyBuffer , p_dtCurrDT , DINT_TO_TIME(p_diCoolTm) , 0 , 1 , 2);

								ELSE
									eStatus	:= Error;

									IF udiStatus = 1000 THEN
										udiStatus	:= 10069;	//Unloading Slot Is Skipped While Unloading Buffer With Cool & Slot Check
									ELSIF udiStatus = 1003 THEN
										udiStatus	:= 10070;	//Unloading Slot Is Not For Board While Unloading Buffer With Cool & Slot Check
									ELSIF udiStatus = 1004 THEN
										udiStatus	:= 10071;	//Unloading Slot Board Is Not available While Unloading Buffer With Cool & Slot Check
									ELSIF udiStatus = 1005 THEN
										udiStatus	:= 10072;	//Unloading Last Sub Slot Is Not For Board While Unloading Buffer With Cool & Slot Check
									ELSIF udiStatus = 1006 THEN
										udiStatus	:= 10073;	//Unloading Last Sub Slot Has No Board While Unloading Buffer With Cool & Slot Check
									ELSIF udiStatus = 1007 THEN
										udiStatus	:= 10074;	//Board Quantity In Slot Is 0 While Unloading Buffer With Cool & Slot Check
									ELSIF udiStatus = 1008 THEN
										udiStatus	:= 10075;	//Board Capacity In Slot Is 0 While Unloading Buffer With Cool & Slot Check
									END_IF

								END_IF

							ELSE
								eStatus	:= Done;

							END_IF

						ELSE
							udiStatus	:= 10035;	//Wrong Slot Number To Unload With Cooling Time Check
							eStatus		:= Error;

						END_IF

					1:
						fbFileWrite1(bEn := TRUE);

						IF fbFileWrite1.udiStatus = 0 THEN
							eStatus	:= Done;
						ELSIF fbFileWrite1.udiStatus < 65534 THEN
							eStatus	:= Error;

							IF fbFileWrite1.udiStatus = 1900 THEN
								udiStatus	:= 10036;	//File Open Error While Unloading Info From Buffer With Slot Check And Cooling Time Check
							ELSIF fbFileWrite1.udiStatus = 1901 THEN
								udiStatus	:= 10037;	//File Create Error While Unloading Info From Buffer With Slot Check And Cooling Time Check
							ELSIF fbFileWrite1.udiStatus = 1903 THEN
								udiStatus	:= 10038;	//File Write Error While Unloading Info From Buffer With Slot Check And Cooling Time Check
							ELSIF fbFileWrite1.udiStatus = 1904 THEN
								udiStatus	:= 10039;	//File Close Error While Unloading Info From Buffer With Slot Check And Cooling Time Check
							ELSIF fbFileWrite1.udiStatus = 1914 THEN
								udiStatus	:= 10047;	//Directory Does Not Exist While Unloading Info From Buffer With Slot Check And Cooling Time Check
							ELSE
								udiStatus	:= fbFileWrite1.udiStatus;
							END_IF
						END_IF

				END_CASE

			END_IF

		BufferActNxtLoad:
			IF eStatus = Idle OR eStatus = Busy THEN

				diCurrSlt	:= fLifterPosInUMToSltBtmMin(p_diLifterCurrPosInUM , p_diSltToSltInUM , p_diLifterBtmPosInUM);

				IF p_bNxtLoadSeq = TRUE THEN
					diNxtLoadSlt	:= fBffrNxtLoadSeqAny(p_bAscending , p_tyBuffer);
				ELSE
					diNxtLoadSlt	:= fBffrNxtLoadNearbyAny(diCurrSlt , p_tyBuffer);
				END_IF

				eStatus	:= Done;

			END_IF

		BufferActNxtLoadGd:
			IF eStatus = Idle OR eStatus = Busy THEN

				diCurrSlt	:= fLifterPosInUMToSltBtmMin(p_diLifterCurrPosInUM , p_diSltToSltInUM , p_diLifterBtmPosInUM);

				IF p_bNxtLoadSeq = TRUE THEN
					diNxtLoadSlt	:= fBffrNxtLoadSeqGd(p_bAscending , p_tyBuffer);
				ELSE
					diNxtLoadSlt	:= fBffrNxtLoadNearbyGd(diCurrSlt , p_tyBuffer);
				END_IF

				eStatus	:= Done;

			END_IF

		BufferActNxtLoadBad:
			IF eStatus = Idle OR eStatus = Busy THEN

				diCurrSlt	:= fLifterPosInUMToSltBtmMin(p_diLifterCurrPosInUM , p_diSltToSltInUM , p_diLifterBtmPosInUM);

				IF p_bNxtLoadSeq = TRUE THEN
					diNxtLoadSlt	:= fBffrNxtLoadSeqBad(p_bAscending , p_tyBuffer);
				ELSE
					diNxtLoadSlt	:= fBffrNxtLoadNearbyBad(diCurrSlt , p_tyBuffer);
				END_IF

				eStatus	:= Done;

			END_IF

		BufferActNxtUnload:
			IF eStatus = Idle OR eStatus = Busy THEN

				IF p_bFIFO = TRUE THEN
					diNxtUnloadSlt	:= fBffrNxtUnloadFIFOAny(p_tyBuffer , '');
				ELSE
					diNxtUnloadSlt	:= fBffrNxtUnloadLIFOAny(p_tyBuffer , '');
				END_IF

				eStatus	:= Done;

			END_IF

		BufferActNxtUnloadGd:
			IF eStatus = Idle OR eStatus = Busy THEN

				IF p_bFIFO = TRUE THEN
					diNxtUnloadSlt	:= fBffrNxtUnloadFIFOGd(p_tyBuffer , '');
				ELSE
					diNxtUnloadSlt	:= fBffrNxtUnloadLIFOGd(p_tyBuffer , '');
				END_IF

				eStatus	:= Done;

			END_IF

		BufferActNxtUnloadBad:
			IF eStatus = Idle OR eStatus = Busy THEN

				IF p_bFIFO = TRUE THEN
					diNxtUnloadSlt	:= fBffrNxtUnloadFIFOBad(p_tyBuffer , '');
				ELSE
					diNxtUnloadSlt	:= fBffrNxtUnloadLIFOBad(p_tyBuffer , '');
				END_IF

				eStatus	:= Done;

			END_IF

		BufferActChkCoolTm:
			diCurrSlt	:= fLifterPosInUMToSltBtmMin(p_diLifterCurrPosInUM , p_diSltToSltInUM , p_diLifterBtmPosInUM);

			bCoolNotRdy	:= NOT fBffrChkCoolTmRdy(diCurrSlt, p_dtCurrDT, DINT_TO_TIME(p_diCoolTm), p_tyBuffer);

			eStatus	:= Done;

		BufferActChkCoolBrdAny:
			diCoolBrdAny	:= fBffrChkCoolBrdAny(p_dtCurrDT, DINT_TO_TIME(p_diCoolTm), p_tyBuffer);

			eStatus	:= Done;

		BufferActChkCoolBrdGd:
			diCoolBrdGd		:= fBffrChkCoolBrdGd(p_dtCurrDT, DINT_TO_TIME(p_diCoolTm), p_tyBuffer);

			eStatus	:= Done;

		BufferActChkCoolBrdBad:
			diCoolBrdBad	:= fBffrChkCoolBrdBad(p_dtCurrDT, DINT_TO_TIME(p_diCoolTm), p_tyBuffer);

			eStatus	:= Done;

		BufferActRstBffr:
			IF eStatus = Idle OR eStatus = Busy THEN

				tyBffrParameter.diBffrTtlSlt	:= p_diBffrTtlSlt;
				tyBffrParameter.diSltCap		:= p_diSltCap;

				memset(ADR(p_tyBuffer) , 0 , SIZEOF(p_tyBuffer));
				fBffrStat(ADR(p_tyBufferStat) , p_tyBuffer);
				fDispBffrDescending(ADR(p_tyDispBuffer) , tyBffrParameter , p_tyBuffer , p_dtCurrDT , DINT_TO_TIME(p_diCoolTm) , 0 , 1 , 2);

				eStatus	:= Done;

			END_IF

		BufferActSetCoolFan:
			IF eStatus = Idle OR eStatus = Busy THEN

				bCoolFanCtrl	:= TRUE;
				eStatus			:= Done;

			END_IF

		BufferActRstCoolFan:
			IF eStatus = Idle OR eStatus = Busy THEN

				bCoolFanCtrl	:= FALSE;
				eStatus			:= Done;

			END_IF

		BufferActBGStartBffrSetFull:
			IF eStatus = Idle OR eStatus = Busy THEN

				bBffrSetFull	:= TRUE;
				bBffrSetMty		:= FALSE;
				eStatus			:= Done;

			END_IF

		BufferActBGStartBffrSetMty:
			IF eStatus = Idle OR eStatus = Busy THEN

				bBffrSetFull	:= FALSE;
				bBffrSetMty		:= TRUE;
				eStatus			:= Done;

			END_IF

		BufferActBGStopBffrSet:
			IF eStatus = Idle OR eStatus = Busy THEN

				bBffrSetFull	:= FALSE;
				bBffrSetMty		:= FALSE;
				eStatus			:= Done;

			END_IF

		BufferActBGStartUpdtSen:
			IF eStatus = Idle OR eStatus = Busy THEN

				bUpdateSensor	:= TRUE;
				eStatus			:= Done;

			END_IF

		BufferActBGStopUpdtSen:
			IF eStatus = Idle OR eStatus = Busy THEN

				bUpdateSensor	:= FALSE;
				eStatus			:= Done;

			END_IF

		BufferActBGStartUpdtDisplay:
			IF eStatus = Idle OR eStatus = Busy THEN

				bUpdtDisplay	:= TRUE;
				eStatus			:= Done;

			END_IF

		BufferActBGStopUpdtDisplay:
			IF eStatus = Idle OR eStatus = Busy THEN

				bUpdtDisplay	:= FALSE;
				eStatus			:= Done;

			END_IF

		BufferActBGStartCoolFan:
			IF eStatus = Idle OR eStatus = Busy THEN

				bCoolFanRun	:= TRUE;
				eStatus		:= Done;

			END_IF

		BufferActBGStopCoolFan:
			IF eStatus = Idle OR eStatus = Busy THEN

				bCoolFanRun	:= FALSE;
				eStatus		:= Done;

			END_IF

	END_CASE

END_ACTION
```

#### Init.st
```iecst
(** 2019-06-07 **)
PROGRAM _INIT

	(* Always Change If Project Change *)

	//Pass Address To Global Address For External Use
	//Action, State & Status
	p_Buffer1Stat		:= ADR(eStat);
	p_Buffer1Status		:= ADR(eStatus);
	p_Buffer1StatTxt	:= ADR(sStatTxt);

	//Alarm
	p_Buffer1AlmData	:= ADR(tyAlmData);

	//Output
	p_Buffer1NxtLoadSlt				:= ADR(diNxtLoadSlt);
	p_Buffer1NxtUnloadSlt			:= ADR(diNxtUnloadSlt);
	p_Buffer1CoolBrdAny				:= ADR(diCoolBrdAny);
	p_Buffer1CoolBrdGd				:= ADR(diCoolBrdGd);
	p_Buffer1CoolBrdBad				:= ADR(diCoolBrdBad);
	p_Buffer1CoolNotRdy				:= ADR(bCoolNotRdy);
	p_Buffer1Bffr					:= ADR(tyBuffer);
	p_Buffer1DispBffr				:= ADR(tyDispBuffer);
	p_Buffer1BffrStat				:= ADR(tyBufferStat);
	p_Buffer1BrdUnloadStat			:= ADR(tyBoardUnloadStat);
	p_Buffer1FileNotFound			:= ADR(bFileNotFound);
	p_Buffer1CoolFanCtrl			:= ADR(bCoolFanCtrl);
	p_Buffer1MagPresent				:= ADR(bMagPresent);
	p_Buffer1MagPresentTm			:= ADR(dtMagPresentTm);
	p_Buffer1NewProduct				:= ADR(bNewProduct);
	p_Buffer1LastProductUnload		:= ADR(bLastProductUnload);
	p_Buffer1LastProductLeftInBffr	:= ADR(bLastProductLeftInBffr);
	p_Buffer1ParamDiff				:= ADR(bParamDiff);
	p_Buffer1MagRemoved				:= ADR(bMagRemoved);
	p_Buffer1FIFOOld				:= ADR(bFIFOOld);

	//Svy Hermes
	p_Buffer1SlotNo					:= ADR(diCurrSltHermes);

	(* Always Change If Project Change *)

END_PROGRAM
```

### Program Logical/Buffer/Buffer2 (IEC) - 1.00.0 - NtBuffer v5.00.0 , NtFileIO v5.00.0

#### InputRef.var
```iecst
(*2019-07-03*)
(**)
(*General*)
VAR
	p_eAct : REFERENCE TO eBufferAction;
	p_udiRstErr : REFERENCE TO UDINT;
END_VAR
(**)
(*Configuration*)
VAR
	p_sFileName : REFERENCE TO STRING[80];
	p_bManual : REFERENCE TO BOOL;
	p_dtCurrDT : REFERENCE TO DATE_AND_TIME;
	p_diMinSlt : REFERENCE TO DINT;
	p_diMaxSlt : REFERENCE TO DINT;
	p_diPitch : REFERENCE TO DINT;
	p_diSltCap : REFERENCE TO DINT;
	p_diBffrTtlSlt : REFERENCE TO DINT;
	p_diCoolTm : REFERENCE TO DINT;
	p_diSltToSltInUM : REFERENCE TO DINT;
	p_diLifterBtmPosInUM : REFERENCE TO DINT;
	p_diLifterCurrPosInUM : REFERENCE TO DINT;
	p_bAscending : REFERENCE TO BOOL;
	p_bFIFO : REFERENCE TO BOOL;
	p_bGdBrdIn : REFERENCE TO BOOL;
	p_bGdBrdReq : REFERENCE TO BOOL;
	p_bNxtLoadSeq : REFERENCE TO BOOL;
	pa_bSkip : REFERENCE TO ARRAY[1..c_diBffrSize] OF BOOL;
	p_diCoolFanOffDlyTm : REFERENCE TO DINT;
	p_bMagPresentSensor : REFERENCE TO BOOL;
	p_bPrepCoolFan : REFERENCE TO BOOL;
	p_bCoolFanTm : REFERENCE TO BOOL;
	p_tyBuffer : REFERENCE TO tyBffr;
	p_tyDispBuffer : REFERENCE TO tyDispBffr;
	p_tyBufferStat : REFERENCE TO tyBffrStat;
	p_sBffrNm : REFERENCE TO STRING[15];
	p_sProdNm : REFERENCE TO STRING[15];
	p_sBarcode1 : REFERENCE TO STRING[80];
	p_sBarcode2 : REFERENCE TO STRING[80];
	p_sCurrRcpNm : REFERENCE TO STRING[15];
	p_sProgNm : REFERENCE TO STRING[15];
	p_bNtSettingsLoadDone : REFERENCE TO BOOL;
END_VAR
```

#### Act_Alarm.st
```iecst
(** 2019-03-25 **)
ACTION Act_Alarm:

	//Error
	IF EDGEPOS(eStatus = Error) THEN

		tyAlmData.sProgNm		:= p_sProgNm;
		tyAlmData.udiCode		:= udiStatus;
		tyAlmData.eSeverity		:= AlmSeverityError;
		tyAlmData.udiRunTime	:= tyAlmData.udiRunTime + 1;
		tyAlmData.bAlm			:= TRUE;
		tyAlmData.udiModuleNum  := udiModuleNum;
		g_sBufferProgNm		:= p_sProgNm;
		//Get Error Message
		IF tyAlmData.udiCode < 10000 OR tyAlmData.udiCode > 10099 THEN
			tyAlmData.sAlmMsg	:= 'Unknown';
			tyAlmData.sRcyMsg	:= 'Unknown';
		ELSE
			tyAlmData.sAlmMsg	:= a_tyAlmText[tyAlmData.udiCode].sAlmText;
			tyAlmData.sRcyMsg	:= a_tyAlmText[tyAlmData.udiCode].sRcyText;
		END_IF

		sStatTxt	:= tyAlmData.sAlmMsg;

	ELSIF bRstErr AND (tyAlmData.udiCode <> 0) THEN

		tyAlmData.udiCode	:= 0;
		tyAlmData.eSeverity	:= AlmSeverityNA;
		tyAlmData.sAlmMsg	:= '';
		tyAlmData.sRcyMsg	:= '';
		tyAlmData.bAlm			:= FALSE;
		sStatTxt	:= a_sStatText[eStat];

	END_IF

END_ACTION
```

#### Act_Background.st
```iecst
(** 2019-07-03 **)
ACTION Act_Background:

	fbMagPresentTm(IN := p_bMagPresentSensor);
	diCurrSltHermes	:= fLifterPosInUMToSltBtmMin(p_diLifterCurrPosInUM , p_diSltToSltInUM , p_diLifterBtmPosInUM);

	//Update Retain
	IF bUpdateSensor = TRUE THEN
		bMagPresent	:= fbMagPresentTm.Q;
	END_IF

	//Display Buffer
	IF bUpdtDisplay = TRUE THEN
		fDispBffrDescending(ADR(p_tyDispBuffer) , tyBffrParameter , p_tyBuffer , p_dtCurrDT , DINT_TO_TIME(p_diCoolTm) , 0 , 1 , 2);
	END_IF

	//Cooling Fan Control
	IF p_bManual = TRUE THEN
		;

	ELSIF bCoolFanRun = TRUE AND p_bPrepCoolFan = TRUE AND bCoolFanTm = TRUE THEN //Cooling Fan Control By Cooling Time

		fbCoolFanOffChkTm(IN := TRUE);

		IF fbCoolFanOffChkTm.Q = TRUE THEN
			IF fBffrChkCoolBrdAny(p_dtCurrDT, DINT_TO_TIME(p_diCoolTm), p_tyBuffer) = 0 THEN
				fbCoolFanOffDlyTm.IN	:= TRUE;
			ELSE
				fbCoolFanOffDlyTm.IN	:= FALSE;
				bCoolFanCtrl			:= TRUE;
			END_IF

			fbCoolFanOffChkTm(IN := FALSE);
		END_IF

		fbCoolFanOffDlyTm;

		IF fbCoolFanOffDlyTm.Q = TRUE THEN
			bCoolFanCtrl	:= FALSE;
		END_IF

	ELSIF bCoolFanRun = TRUE AND p_bPrepCoolFan = TRUE AND bCoolFanTm = FALSE THEN	//Cooling Fan Control By Buffer Empty
		fbCoolFanOffDlyTm(IN := p_tyBufferStat.bBffrMty);

		IF p_tyBufferStat.bBffrMty = FALSE THEN
			bCoolFanCtrl	:= TRUE;
		END_IF

		IF fbCoolFanOffDlyTm.Q = TRUE THEN
			bCoolFanCtrl	:= FALSE;
		END_IF

	ELSE

		bCoolFanCtrl	:= FALSE;

	END_IF

	//Set Buffer By Magazine Present
	IF bBffrSetFull = TRUE THEN
		IF p_bMagPresentSensor = TRUE AND fbMagAbsentTm.Q = TRUE THEN
			bSetFull		:= TRUE;
			dtMagPresentTm	:= p_dtCurrDT;
		END_IF

		IF bSetFull = TRUE THEN
			p_eAct	:= BufferActSetFull;

			IF eStatus = Done AND eStat = BufferActSetFull THEN
				p_eAct		:= BufferActIdle;
				bSetFull	:= FALSE;
			ELSIF eStatus = Error THEN
				bSetFull	:= FALSE;
			END_IF
		END_IF

		fbMagAbsentTm(IN := NOT p_bMagPresentSensor);

	ELSIF bBffrSetMty = TRUE THEN
		IF p_bMagPresentSensor = TRUE AND fbMagAbsentTm.Q = TRUE THEN
			bSetMty			:= TRUE;
			dtMagPresentTm	:= p_dtCurrDT;
		END_IF

		IF bSetMty = TRUE THEN
			p_eAct	:= BufferActSetMty;

			IF eStatus = Done AND eStat = BufferActSetMty THEN
				p_eAct	:= BufferActIdle;
				bSetMty	:= FALSE;
			ELSIF eStatus = Error THEN
				bSetMty	:= FALSE;
			END_IF
		END_IF

		fbMagAbsentTm(IN := NOT p_bMagPresentSensor);

	END_IF

	//Check Parameter Different
	bParamDiff	:= (tyBffrParameter.bAscending <> p_bAscending)
	OR (tyBffrParameter.diMinSlt <> p_diMinSlt)
	OR (tyBffrParameter.diMaxSlt <> p_diMaxSlt)
	OR (tyBffrParameter.diPitch <> p_diPitch)
	OR (tyBffrParameter.diSltCap <> p_diSltCap)
	OR (bFIFOOld <> p_bFIFO);

	//Update MagRemoved
	bMagRemoved	:= fbMagAbsentTm.Q;

END_ACTION
```

#### Act_InitGlobal.st
```iecst
(** 2019-04-26 **)
ACTION Act_InitGlobal:

	(* Always Change If Project Change *)

	//Pass Data To Link
	p_bLinkStartupRun ACCESS p_StartupRun;
	p_bLinkNtParamProjMagConvPrep ACCESS p_NtParamProjMag2ConvPrep;
//	p_eLinkOpsMagLDBufferAct ACCESS p_OpsMagLD2BufferAct;
	p_eLinkOpsMagConvLDBufferAct ACCESS p_OpsMagConvLD2BufferAct;

	p_bLinkMcParamProdSelTopToBtm ACCESS p_NtParamProjTopToBtmDefault;//p_ProdRcpCurrRcp1TopToBtm;
	p_bLinkPresentSen1 ACCESS p_DIMagPresentSen2;
	p_bLinkPresentSen2 ACCESS p_DIMagConvEntSen2;

	p_eLinkMag ACCESS p_NtParamProjMag;
	p_usiLinkMod ACCESS p_ProdRcpCurrRcp1McMod;

	p_diLinkSltToSltDist ACCESS p_MagRcpCurrRcpSltToSlt;
	p_diLinkMinSlt ACCESS p_ProdRcpCurrRcp1MinSltValue;
	p_diLinkMaxSlt ACCESS p_ProdRcpCurrRcp1MaxSltValue;
	p_diLinkPitch ACCESS p_ProdRcpCurrRcp1Pitch;
	p_diLinkBffrTtlSlt ACCESS p_MagRcpCurrRcpTtlSlt;
	p_diLinkLifterBtmPosInUM ACCESS p_MagRcpCurrRcpMag2Slt1Pos;

	p_diLinkSltToSltDist1 ACCESS p_MagRcpCurrRcpSltToSlt1;
	p_diLinkMinSlt1 ACCESS p_ProdRcpCurrRcp1MinSltRear;
	p_diLinkMaxSlt1 ACCESS p_ProdRcpCurrRcp1MaxSltRear;
	p_diLinkPitch1 ACCESS p_ProdRcpCurrRcp1PitchRear;
	p_diLinkBffrTtlSlt1 ACCESS p_MagRcpCurrRcpTtlSlt1;
	p_diLinkLifterBtmPosInUM1 ACCESS p_MagRcpCurrRcpMag2Slt1Pos1;

	p_bLinkNtParamProjRotCylPrep ACCESS p_NtParamProjPullerRotCylPrep;

	p_bLinkProjLifterMagPlatform ACCESS p_NtParamProjLifterMagPlatform;
	p_diNtParamProjMagMaxSlt ACCESS p_NtParamProjMagMaxSlt; //initial
	p_eLinkOpsLifMagLDBufferAct ACCESS p_OpsLifMagLDBufferAct2;
	p_bNtParamAutoRcpPrep ACCESS p_NtParamAutoRcpPrep;
	p_bHermesSvyPrep ACCESS p_NtParamHermesSvyPrep; //queryWO
	p_bMcParamHermesSvyEn ACCESS p_McParamHermesSvyEn;
	p_eNtParamCustomerReq ACCESS p_NtParamCustomerReq;
	p_bMcParamMesRFIDEn ACCESS p_McParamMesRFIDEn;

	//Pass Data To Internal Use
	p_udiRstErr ACCESS p_RstErrReset;
	p_sFileName ACCESS p_NtParamBffr2FileNm;
	p_bManual ACCESS p_UIMnlMod;
	p_dtCurrDT ACCESS p_TimeCurrDT;
//	p_diMinSlt ACCESS p_ProdRcpCurrRcp1MinSltValue;
//	p_diMaxSlt ACCESS p_ProdRcpCurrRcp1MaxSltValue;
//	p_diPitch ACCESS p_ProdRcpCurrRcp1Pitch;
//	p_diBffrTtlSlt ACCESS p_MagRcpCurrRcpTtlSlt;
//	p_diLifterBtmPosInUM ACCESS p_MagRcpCurrRcpMag2Slt1Pos;
	p_diLifterCurrPosInUM ACCESS p_LifterBtmActualPos;
	p_bFIFO ACCESS p_NtParamBffr2FIFO;
//	p_bMagPresentSensor ACCESS p_DIMagPresentSen2;
	p_sCurrRcpNm ACCESS p_ProdRcpCurrRcp1Nm;
	p_sProgNm ACCESS p_NtParamBffr2ProgNm;
	p_bNtSettingsLoadDone ACCESS p_StartupNtSettingsLoadDone;

	(* Always Change If Project Change *)

END_ACTION
```

#### Act_Link.st
```iecst
(** 2019-03-29 **)
ACTION Act_Link:

	IF p_eLinkMag = LDMagQuadruple THEN
		CASE p_usiLinkMod OF
			0,2: //LDModLoadLnA, LDModLoadLnAB:
				IF p_bAscending THEN
					p_diSltToSltInUM := p_diLinkSltToSltDist * -1;
				ELSE
					p_diSltToSltInUM := p_diLinkSltToSltDist;
				END_IF
				p_diMinSlt := p_diLinkMinSlt;
				p_diMaxSlt := p_diLinkMaxSlt;
				p_diPitch := p_diLinkPitch;
				p_diBffrTtlSlt := p_diLinkBffrTtlSlt;
				p_diLifterBtmPosInUM := p_diLinkLifterBtmPosInUM;

			1: //LDModLoadLnB:
				IF p_bAscending THEN
					p_diSltToSltInUM := p_diLinkSltToSltDist1 * -1;
				ELSE
					p_diSltToSltInUM := p_diLinkSltToSltDist1;
				END_IF
				p_diSltToSltInUM := p_diLinkSltToSltDist1;
				p_diMinSlt := p_diLinkMinSlt1;
				p_diMaxSlt := p_diLinkMaxSlt1;
				p_diPitch := p_diLinkPitch1;
				p_diBffrTtlSlt := p_diLinkBffrTtlSlt1;
				p_diLifterBtmPosInUM := p_diLinkLifterBtmPosInUM1;

		END_CASE
	ELSE
		IF p_bAscending THEN
			p_diSltToSltInUM := p_diLinkSltToSltDist * -1;
		ELSE
			p_diSltToSltInUM := p_diLinkSltToSltDist;
		END_IF
		IF p_bNtParamAutoRcpPrep AND ((p_bHermesSvyPrep AND p_bMcParamHermesSvyEn) OR (p_eNtParamCustomerReq = We_Fabricate AND p_bMcParamMesRFIDEn)) THEN
			p_diMinSlt ACCESS p_diAutoRcpMag2MinSlt;
			p_diMaxSlt ACCESS p_diAutoRcpMag2MaxSlt;
			p_diPitch ACCESS p_diAutoRcpMag2Pitch;
		ELSE
			p_diMinSlt ACCESS ADR(diMinSlt);
			p_diMaxSlt ACCESS ADR(diMaxSlt);
			p_diPitch ACCESS ADR(diPitch);
			p_diMinSlt := p_diLinkMinSlt;
			p_diMaxSlt := p_diLinkMaxSlt;
			p_diPitch := p_diLinkPitch;
		END_IF
		p_diBffrTtlSlt := p_diLinkBffrTtlSlt;
		p_diLifterBtmPosInUM := p_diLinkLifterBtmPosInUM;
	END_IF

	p_bAscending	:= NOT p_bLinkMcParamProdSelTopToBtm;
//	IF p_bLinkNtParamProjRotCylPrep THEN
//		p_bAscending := TRUE;
//	ELSE
//		p_bAscending := FALSE;
//	END_IF

	IF p_bLinkNtParamProjMagConvPrep THEN
		fbMagPresentTm.PT	:= T#2s;
	ELSE
		fbMagPresentTm.PT	:= T#8s;
	END_IF

	p_bMagPresentSensor := p_bLinkPresentSen1 OR p_bLinkPresentSen2;

END_ACTION
```

#### Act_LinkAction.st
```iecst
(** 2019-05-10 **)
ACTION Act_LinkAction:

	IF p_bLinkStartupRun = TRUE THEN
		p_eAct ACCESS p_StartupBuffer2Act;
	ELSE
		IF eStatus = Idle THEN
			IF p_bLinkProjLifterMagPlatform = FALSE THEN
				IF p_eLinkOpsMagConvLDBufferAct <> BufferActIdle THEN
					p_eAct ACCESS p_OpsMagConvLD2BufferAct;
				ELSE
					p_eAct ACCESS p_UIBuffer2Act;
				END_IF
			ELSE
				IF p_eLinkOpsLifMagLDBufferAct <> BufferActIdle THEN
					p_eAct ACCESS p_OpsLifMagLDBufferAct2;
				ELSE
					p_eAct ACCESS p_UIBuffer2Act;
				END_IF
			END_IF
		END_IF
	END_IF

END_ACTION
```
